LIN {X 0,Y 481.22,Z 200.296,A -85,B 0,C 180,E1 -6765.441,E2 -6765.441} C_VEL
LIN {X 0,Y 481.227,Z 196.018,A -85,B 0,C 180,E1 -6768.74,E2 -6768.74} C_VEL
LIN {X 0,Y 481.265,Z 192.611,A -85,B 0,C 180,E1 -6771.411,E2 -6771.411} C_VEL
LIN {X 0,Y 481.352,Z 189.237,A -85,B 0,C 180,E1 -6774.129,E2 -6774.129} C_VEL
LIN {X 0,Y 481.456,Z 185.54,A -85,B 0,C 180,E1 -6777.071,E2 -6777.071} C_VEL
LIN {X 0,Y 481.476,Z 183.514,A -85,B 0,C 180,E1 -6778.859,E2 -6778.859} C_VEL
LIN {X 0,Y 481.635,Z 183.493,A -85,B 0,C 180,E1 -6781.688,E2 -6781.688} C_VEL
LIN {X 0,Y 481.688,Z 183.482,A -85,B 0,C 180,E1 -6784.681,E2 -6784.681} C_VEL
LIN {X 0,Y 481.651,Z 183.487,A -85,B 0,C 180,E1 -6788.006,E2 -6788.006} C_VEL
LIN {X 0,Y 481.657,Z 183.49,A -85,B 0,C 180,E1 -6791.04,E2 -6791.04} C_VEL
LIN {X 0,Y 481.652,Z 183.484,A -85,B 0,C 180,E1 -6794.358,E2 -6794.358} C_VEL
LIN {X 0,Y 481.637,Z 183.492,A -85,B 0,C 180,E1 -6796.85,E2 -6796.85} C_VEL
LIN {X 0,Y 481.677,Z 183.481,A -85,B 0,C 180,E1 -6800.059,E2 -6800.059} C_VEL
LIN {X 0,Y 481.625,Z 183.488,A -85,B 0,C 180,E1 -6803.374,E2 -6803.374} C_VEL
LIN {X 0,Y 481.701,Z 183.482,A -85,B 0,C 180,E1 -6806.329,E2 -6806.329} C_VEL
LIN {X 0,Y 481.649,Z 183.484,A -85,B 0,C 180,E1 -6809.415,E2 -6809.415} C_VEL
LIN {X 0,Y 481.693,Z 183.485,A -85,B 0,C 180,E1 -6812.167,E2 -6812.167} C_VEL
LIN {X 0,Y 481.708,Z 183.474,A -85,B 0,C 180,E1 -6814.969,E2 -6814.969} C_VEL
LIN {X 0,Y 481.643,Z 183.49,A -85,B 0,C 180,E1 -6817.704,E2 -6817.704} C_VEL
LIN {X 0,Y 481.698,Z 183.479,A -85,B 0,C 180,E1 -6820.393,E2 -6820.393} C_VEL
LIN {X 0,Y 481.681,Z 183.482,A -85,B 0,C 180,E1 -6823.033,E2 -6823.033} C_VEL
LIN {X 0,Y 481.679,Z 183.484,A -85,B 0,C 180,E1 -6825.638,E2 -6825.638} C_VEL
LIN {X 0,Y 481.741,Z 183.473,A -85,B 0,C 180,E1 -6828.215,E2 -6828.215} C_VEL
LIN {X 0,Y 481.753,Z 183.476,A -85,B 0,C 180,E1 -6831.611,E2 -6831.611} C_VEL
LIN {X 0,Y 481.797,Z 183.464,A -85,B 0,C 180,E1 -6834.139,E2 -6834.139} C_VEL
LIN {X 0,Y 481.915,Z 183.454,A -85,B 0,C 180,E1 -6837.492,E2 -6837.492} C_VEL
LIN {X 0,Y 481.894,Z 183.456,A -85,B 0,C 180,E1 -6840.836,E2 -6840.836} C_VEL
LIN {X 0,Y 481.913,Z 183.455,A -85,B 0,C 180,E1 -6842.507,E2 -6842.507} C_VEL
LIN {X 0,Y 481.793,Z 183.466,A -85,B 0,C 180,E1 -6845.861,E2 -6845.861} C_VEL
LIN {X 0,Y 481.749,Z 183.478,A -85,B 0,C 180,E1 -6848.389,E2 -6848.389} C_VEL
LIN {X 0,Y 481.738,Z 183.475,A -85,B 0,C 180,E1 -6851.785,E2 -6851.785} C_VEL
LIN {X 0,Y 481.73,Z 183.475,A -85,B 0,C 180,E1 -6855.225,E2 -6855.225} C_VEL
LIN {X 0,Y 481.695,Z 183.481,A -85,B 0,C 180,E1 -6858.722,E2 -6858.722} C_VEL
LIN {X 0,Y 481.632,Z 183.489,A -85,B 0,C 180,E1 -6861.395,E2 -6861.395} C_VEL
LIN {X 0,Y 481.636,Z 183.493,A -85,B 0,C 180,E1 -6864.115,E2 -6864.115} C_VEL
LIN {X 0,Y 481.639,Z 183.489,A -85,B 0,C 180,E1 -6867.117,E2 -6867.117} C_VEL
LIN {X 0,Y 481.654,Z 183.491,A -85,B 0,C 180,E1 -6869.743,E2 -6869.743} C_VEL
LIN {X 0,Y 481.66,Z 183.484,A -85,B 0,C 180,E1 -6872.675,E2 -6872.675} C_VEL
LIN {X 0,Y 481.621,Z 183.493,A -85,B 0,C 180,E1 -6875.711,E2 -6875.711} C_VEL
LIN {X 0,Y 481.656,Z 183.491,A -85,B 0,C 180,E1 -6878.861,E2 -6878.861} C_VEL
LIN {X 0,Y 481.632,Z 183.489,A -85,B 0,C 180,E1 -6882.163,E2 -6882.163} C_VEL
LIN {X 0,Y 481.647,Z 183.488,A -85,B 0,C 180,E1 -6885.543,E2 -6885.543} C_VEL
LIN {X 0,Y 481.649,Z 183.492,A -85,B 0,C 180,E1 -6888.959,E2 -6888.959} C_VEL
LIN {X 0,Y 481.649,Z 183.49,A -85,B 0,C 180,E1 -6891.994,E2 -6891.994} C_VEL
LIN {X 0,Y 481.685,Z 183.481,A -85,B 0,C 180,E1 -6895.319,E2 -6895.319} C_VEL
LIN {X 0,Y 481.73,Z 183.66,A -85,B 0,C 180,E1 -6895.956,E2 -6895.956} C_VEL
LIN {X 0,Y 484.668,Z 196.394,A -85,B 0,C 180,E1 -6898.82,E2 -6898.82} C_VEL
LIN {X 0,Y 485.724,Z 201.979,A -85,B 0,C 180,E1 -6899.982,E2 -6899.982} C_VEL
LIN {X 0,Y 484.86,Z 216.213,A -85,B 0,C 180,E1 -6902.601,E2 -6902.601} C_VEL
LIN {X 0,Y 483.78,Z 235.626,A -85,B 0,C 180,E1 -6906,E2 -6906} C_VEL
LIN {X 0,Y 482.882,Z 255.103,A -85,B 0,C 180,E1 -6909.334,E2 -6909.334} C_VEL
LIN {X 0,Y 482.267,Z 271.753,A -85,B 0,C 180,E1 -6912.181,E2 -6912.181} C_VEL
LIN {X 0,Y 481.736,Z 289.457,A -85,B 0,C 180,E1 -6915.264,E2 -6915.264} C_VEL
LIN {X 0,Y 483.157,Z 305.726,A -85,B 0,C 180,E1 -6915.658,E2 -6915.658} C_VEL
LIN {X 0,Y 483.299,Z 312.328,A -85,B 0,C 180,E1 -6915.877,E2 -6915.877} C_VEL
LIN {X 0,Y 482.991,Z 325.423,A -85,B 0,C 180,E1 -6916.431,E2 -6916.431} C_VEL
LIN {X 0,Y 482.648,Z 336.61,A -85,B 0,C 180,E1 -6917.064,E2 -6917.064} C_VEL
LIN {X 0,Y 482.217,Z 348.057,A -85,B 0,C 180,E1 -6917.898,E2 -6917.898} C_VEL
LIN {X 0,Y 481.899,Z 358.618,A -85,B 0,C 180,E1 -6918.859,E2 -6918.859} C_VEL
LIN {X 0,Y 481.535,Z 368.02,A -85,B 0,C 180,E1 -6919.914,E2 -6919.914} C_VEL
LIN {X 0,Y 481.3,Z 377.093,A -85,B 0,C 180,E1 -6921.182,E2 -6921.182} C_VEL
LIN {X 0,Y 481.122,Z 384.382,A -85,B 0,C 180,E1 -6922.447,E2 -6922.447} C_VEL
LIN {X 0,Y 480.978,Z 390.38,A -85,B 0,C 180,E1 -6923.765,E2 -6923.765} C_VEL
LIN {X 0,Y 481.008,Z 394.686,A -85,B 0,C 180,E1 -6924.972,E2 -6924.972} C_VEL
LIN {X 0,Y 481.023,Z 397.058,A -85,B 0,C 180,E1 -6925.812,E2 -6925.812} C_VEL
LIN {X 0,Y 481.004,Z 398.985,A -85,B 0,C 180,E1 -6926.651,E2 -6926.651} C_VEL
LIN {X 0,Y 481.007,Z 400.451,A -85,B 0,C 180,E1 -6927.489,E2 -6927.489} C_VEL
LIN {X 0,Y 480.932,Z 402.075,A -85,B 0,C 180,E1 -6929.164,E2 -6929.164} C_VEL
LIN {X 0,Y 480.947,Z 402.282,A -85,B 0,C 180,E1 -6930.001,E2 -6930.001} C_VEL
LIN {X 0,Y 480.933,Z 402.03,A -85,B 0,C 180,E1 -6930.838,E2 -6930.838} C_VEL
LIN {X 0,Y 480.944,Z 401.367,A -85,B 0,C 180,E1 -6931.676,E2 -6931.676} C_VEL
LIN {X 0,Y 481.01,Z 400.303,A -85,B 0,C 180,E1 -6932.513,E2 -6932.513} C_VEL
LIN {X 0,Y 481.029,Z 398.792,A -85,B 0,C 180,E1 -6933.351,E2 -6933.351} C_VEL
LIN {X 0,Y 480.999,Z 395.665,A -85,B 0,C 180,E1 -6934.61,E2 -6934.61} C_VEL
LIN {X 0,Y 481.021,Z 391.432,A -85,B 0,C 180,E1 -6935.871,E2 -6935.871} C_VEL
LIN {X 0,Y 481.122,Z 384.92,A -85,B 0,C 180,E1 -6937.344,E2 -6937.344} C_VEL
LIN {X 0,Y 481.279,Z 377.82,A -85,B 0,C 180,E1 -6938.609,E2 -6938.609} C_VEL
LIN {X 0,Y 481.465,Z 368.907,A -85,B 0,C 180,E1 -6939.877,E2 -6939.877} C_VEL
LIN {X 0,Y 481.857,Z 358.791,A -85,B 0,C 180,E1 -6941.037,E2 -6941.037} C_VEL
LIN {X 0,Y 482.137,Z 347.375,A -85,B 0,C 180,E1 -6942.079,E2 -6942.079} C_VEL
LIN {X 0,Y 482.567,Z 335.494,A -85,B 0,C 180,E1 -6942.94,E2 -6942.94} C_VEL
LIN {X 0,Y 482.965,Z 323.218,A -85,B 0,C 180,E1 -6943.625,E2 -6943.625} C_VEL
LIN {X 0,Y 483.345,Z 309.934,A -85,B 0,C 180,E1 -6944.178,E2 -6944.178} C_VEL
LIN {X 0,Y 482.359,Z 295.934,A -85,B 0,C 180,E1 -6944.598,E2 -6944.598} C_VEL
LIN {X 0,Y 481.731,Z 289.296,A -85,B 0,C 180,E1 -6944.766,E2 -6944.766} C_VEL
LIN {X 0,Y 482.271,Z 270.473,A -85,B 0,C 180,E1 -6948.04,E2 -6948.04} C_VEL
LIN {X 0,Y 483.142,Z 250.047,A -85,B 0,C 180,E1 -6951.527,E2 -6951.527} C_VEL
LIN {X 0,Y 483.948,Z 231.674,A -85,B 0,C 180,E1 -6954.679,E2 -6954.679} C_VEL
LIN {X 0,Y 485.004,Z 213.512,A -85,B 0,C 180,E1 -6957.88,E2 -6957.88} C_VEL
LIN {X 0,Y 485.715,Z 201.921,A -85,B 0,C 180,E1 -6960.02,E2 -6960.02} C_VEL
LIN {X 0,Y 484.026,Z 193.683,A -85,B 0,C 180,E1 -6961.76,E2 -6961.76} C_VEL
LIN {X 0,Y 481.676,Z 183.492,A -85,B 0,C 180,E1 -6964.114,E2 -6964.114} C_VEL
LIN {X 0,Y 481.624,Z 183.496,A -85,B 0,C 180,E1 -6966.748,E2 -6966.748} C_VEL
LIN {X 0,Y 481.68,Z 183.486,A -85,B 0,C 180,E1 -6969.941,E2 -6969.941} C_VEL
LIN {X 0,Y 481.643,Z 183.49,A -85,B 0,C 180,E1 -6973.3,E2 -6973.3} C_VEL
LIN {X 0,Y 481.659,Z 183.491,A -85,B 0,C 180,E1 -6975.642,E2 -6975.642} C_VEL
LIN {X 0,Y 481.661,Z 183.491,A -85,B 0,C 180,E1 -6978.959,E2 -6978.959} C_VEL
LIN {X 0,Y 481.652,Z 183.49,A -85,B 0,C 180,E1 -6981.994,E2 -6981.994} C_VEL
LIN {X 0,Y 481.656,Z 183.504,A -85,B 0,C 180,E1 -6984.434,E2 -6984.434} C_VEL
LIN {X 0,Y 482.299,Z 187.95,A -85,B 0,C 180,E1 -6985.818,E2 -6985.818} C_VEL
LIN {X 0,Y 482.217,Z 196.061,A -85,B 0,C 180,E1 -6988.353,E2 -6988.353} C_VEL
LIN {X 0,Y 482.096,Z 206.422,A -85,B 0,C 180,E1 -6991.72,E2 -6991.72} C_VEL
LIN {X 0,Y 481.964,Z 215.165,A -85,B 0,C 180,E1 -6994.701,E2 -6994.701} C_VEL
LIN {X 0,Y 481.919,Z 222.689,A -85,B 0,C 180,E1 -6997.266,E2 -6997.266} C_VEL
LIN {X 0,Y 481.814,Z 231.6,A -85,B 0,C 180,E1 -7000.398,E2 -7000.398} C_VEL
LIN {X 0,Y 481.648,Z 241.418,A -85,B 0,C 180,E1 -7003.904,E2 -7003.904} C_VEL
LIN {X 0,Y 481.627,Z 244.929,A -85,B 0,C 180,E1 -7005.151,E2 -7005.151} C_VEL
LIN {X 0,Y 484.117,Z 257.015,A -85,B 0,C 180,E1 -7005.578,E2 -7005.578} C_VEL
LIN {X 0,Y 483.742,Z 270.706,A -85,B 0,C 180,E1 -7006.13,E2 -7006.13} C_VEL
LIN {X 0,Y 483.373,Z 283.042,A -85,B 0,C 180,E1 -7006.816,E2 -7006.816} C_VEL
LIN {X 0,Y 482.982,Z 295.454,A -85,B 0,C 180,E1 -7007.713,E2 -7007.713} C_VEL
LIN {X 0,Y 482.514,Z 305.818,A -85,B 0,C 180,E1 -7008.66,E2 -7008.66} C_VEL
LIN {X 0,Y 482.131,Z 315.197,A -85,B 0,C 180,E1 -7009.714,E2 -7009.714} C_VEL
LIN {X 0,Y 481.808,Z 322.924,A -85,B 0,C 180,E1 -7010.767,E2 -7010.767} C_VEL
LIN {X 0,Y 481.491,Z 330.49,A -85,B 0,C 180,E1 -7012.029,E2 -7012.029} C_VEL
LIN {X 0,Y 481.263,Z 337.504,A -85,B 0,C 180,E1 -7013.525,E2 -7013.525} C_VEL
LIN {X 0,Y 480.997,Z 342.655,A -85,B 0,C 180,E1 -7014.971,E2 -7014.971} C_VEL
LIN {X 0,Y 481.068,Z 344.937,A -85,B 0,C 180,E1 -7015.811,E2 -7015.811} C_VEL
LIN {X 0,Y 481.003,Z 346.806,A -85,B 0,C 180,E1 -7016.649,E2 -7016.649} C_VEL
LIN {X 0,Y 480.947,Z 348.246,A -85,B 0,C 180,E1 -7017.487,E2 -7017.487} C_VEL
LIN {X 0,Y 480.772,Z 349.845,A -85,B 0,C 180,E1 -7019.162,E2 -7019.162} C_VEL
LIN {X 0,Y 480.759,Z 350.06,A -85,B 0,C 180,E1 -7020,E2 -7020} C_VEL
LIN {X 0,Y 480.77,Z 349.843,A -85,B 0,C 180,E1 -7020.838,E2 -7020.838} C_VEL
LIN {X 0,Y 480.945,Z 348.202,A -85,B 0,C 180,E1 -7022.513,E2 -7022.513} C_VEL
LIN {X 0,Y 480.991,Z 346.783,A -85,B 0,C 180,E1 -7023.351,E2 -7023.351} C_VEL
LIN {X 0,Y 481.03,Z 343.822,A -85,B 0,C 180,E1 -7024.609,E2 -7024.609} C_VEL
LIN {X 0,Y 481.155,Z 339.808,A -85,B 0,C 180,E1 -7025.869,E2 -7025.869} C_VEL
LIN {X 0,Y 481.287,Z 334.625,A -85,B 0,C 180,E1 -7027.13,E2 -7027.13} C_VEL
LIN {X 0,Y 481.524,Z 328.112,A -85,B 0,C 180,E1 -7028.393,E2 -7028.393} C_VEL
LIN {X 0,Y 481.826,Z 320.026,A -85,B 0,C 180,E1 -7029.657,E2 -7029.657} C_VEL
LIN {X 0,Y 482.145,Z 311.758,A -85,B 0,C 180,E1 -7030.711,E2 -7030.711} C_VEL
LIN {X 0,Y 482.577,Z 301.598,A -85,B 0,C 180,E1 -7031.765,E2 -7031.765} C_VEL
LIN {X 0,Y 483.004,Z 290.302,A -85,B 0,C 180,E1 -7032.712,E2 -7032.712} C_VEL
LIN {X 0,Y 483.372,Z 279.109,A -85,B 0,C 180,E1 -7033.452,E2 -7033.452} C_VEL
LIN {X 0,Y 483.784,Z 266.716,A -85,B 0,C 180,E1 -7034.083,E2 -7034.083} C_VEL
LIN {X 0,Y 483.821,Z 255.619,A -85,B 0,C 180,E1 -7034.512,E2 -7034.512} C_VEL
LIN {X 0,Y 481.407,Z 243.352,A -85,B 0,C 180,E1 -7034.937,E2 -7034.937} C_VEL
LIN {X 0,Y 481.526,Z 235.352,A -85,B 0,C 180,E1 -7037.849,E2 -7037.849} C_VEL
LIN {X 0,Y 481.658,Z 226.855,A -85,B 0,C 180,E1 -7040.957,E2 -7040.957} C_VEL
LIN {X 0,Y 481.787,Z 219.5,A -85,B 0,C 180,E1 -7043.65,E2 -7043.65} C_VEL
LIN {X 0,Y 481.951,Z 210.681,A -85,B 0,C 180,E1 -7046.876,E2 -7046.876} C_VEL
LIN {X 0,Y 482.102,Z 202.963,A -85,B 0,C 180,E1 -7049.713,E2 -7049.713} C_VEL
LIN {X 0,Y 482.175,Z 195.007,A -85,B 0,C 180,E1 -7052.636,E2 -7052.636} C_VEL
LIN {X 0,Y 482.255,Z 187.65,A -85,B 0,C 180,E1 -7055.303,E2 -7055.303} C_VEL
LIN {X 0,Y 481.664,Z 183.489,A -85,B 0,C 180,E1 -7056.874,E2 -7056.874} C_VEL
LIN {X 0,Y 481.664,Z 183.487,A -85,B 0,C 180,E1 -7059.942,E2 -7059.942} C_VEL
LIN {X 0,Y 481.632,Z 183.491,A -85,B 0,C 180,E1 -7063.146,E2 -7063.146} C_VEL
LIN {X 0,Y 481.659,Z 183.487,A -85,B 0,C 180,E1 -7065.641,E2 -7065.641} C_VEL
LIN {X 0,Y 481.662,Z 183.49,A -85,B 0,C 180,E1 -7068.958,E2 -7068.958} C_VEL
LIN {X 0,Y 481.638,Z 183.492,A -85,B 0,C 180,E1 -7071.996,E2 -7071.996} C_VEL
LIN {X 0,Y 481.684,Z 183.488,A -85,B 0,C 180,E1 -7075.317,E2 -7075.317} C_VEL
LIN {X 0,Y 481.644,Z 183.49,A -85,B 0,C 180,E1 -7078.311,E2 -7078.311} C_VEL
LIN {X 0,Y 481.5,Z 183.509,A -85,B 0,C 180,E1 -7080.719,E2 -7080.719} C_VEL
LIN {X 0,Y 480.796,Z 183.851,A -85,B 0,C 180,E1 -7081.415,E2 -7081.415} C_VEL
LIN {X 0,Y 477.902,Z 185.342,A -85,B 0,C 180,E1 -7082.535,E2 -7082.535} C_VEL
LIN {X 0,Y 475.475,Z 186.77,A -85,B 0,C 180,E1 -7083.435,E2 -7083.435} C_VEL
LIN {X 0,Y 474.442,Z 187.776,A -85,B 0,C 180,E1 -7084.131,E2 -7084.131} C_VEL
LIN {X 0,Y 474.362,Z 188.066,A -85,B 0,C 180,E1 -7084.368,E2 -7084.368} C_VEL
LIN {X 0,Y 474.254,Z 191.754,A -85,B 0,C 180,E1 -7087.337,E2 -7087.337} C_VEL
LIN {X 0,Y 474.182,Z 195.164,A -85,B 0,C 180,E1 -7090.068,E2 -7090.068} C_VEL
LIN {X 0,Y 474.127,Z 198.642,A -85,B 0,C 180,E1 -7092.754,E2 -7092.754} C_VEL
LIN {X 0,Y 474.114,Z 202.159,A -85,B 0,C 180,E1 -7095.403,E2 -7095.403} C_VEL
LIN {X 0,Y 474.212,Z 205.883,A -85,B 0,C 180,E1 -7098.024,E2 -7098.024} C_VEL
LIN {X 0,Y 474.137,Z 209.896,A -85,B 0,C 180,E1 -7100.642,E2 -7100.642} C_VEL
LIN {X 0,Y 476.144,Z 219.9,A -85,B 0,C 180,E1 -7101.083,E2 -7101.083} C_VEL
LIN {X 0,Y 476.003,Z 228.87,A -85,B 0,C 180,E1 -7101.585,E2 -7101.585} C_VEL
LIN {X 0,Y 475.902,Z 236.501,A -85,B 0,C 180,E1 -7102.162,E2 -7102.162} C_VEL
LIN {X 0,Y 475.649,Z 242.928,A -85,B 0,C 180,E1 -7102.784,E2 -7102.784} C_VEL
LIN {X 0,Y 475.534,Z 249.697,A -85,B 0,C 180,E1 -7103.635,E2 -7103.635} C_VEL
LIN {X 0,Y 475.19,Z 255.993,A -85,B 0,C 180,E1 -7104.695,E2 -7104.695} C_VEL
LIN {X 0,Y 475.005,Z 260.57,A -85,B 0,C 180,E1 -7105.756,E2 -7105.756} C_VEL
LIN {X 0,Y 474.731,Z 264.378,A -85,B 0,C 180,E1 -7107.029,E2 -7107.029} C_VEL
LIN {X 0,Y 474.572,Z 266.665,A -85,B 0,C 180,E1 -7108.302,E2 -7108.302} C_VEL
LIN {X 0,Y 474.49,Z 267.471,A -85,B 0,C 180,E1 -7109.15,E2 -7109.15} C_VEL
LIN {X 0,Y 474.459,Z 267.751,A -85,B 0,C 180,E1 -7109.999,E2 -7109.999} C_VEL
LIN {X 0,Y 474.482,Z 267.526,A -85,B 0,C 180,E1 -7110.848,E2 -7110.848} C_VEL
LIN {X 0,Y 474.521,Z 266.784,A -85,B 0,C 180,E1 -7111.696,E2 -7111.696} C_VEL
LIN {X 0,Y 474.576,Z 265.484,A -85,B 0,C 180,E1 -7112.545,E2 -7112.545} C_VEL
LIN {X 0,Y 474.921,Z 262.316,A -85,B 0,C 180,E1 -7113.817,E2 -7113.817} C_VEL
LIN {X 0,Y 475.055,Z 257.48,A -85,B 0,C 180,E1 -7115.091,E2 -7115.091} C_VEL
LIN {X 0,Y 475.298,Z 253.005,A -85,B 0,C 180,E1 -7115.94,E2 -7115.94} C_VEL
LIN {X 0,Y 475.509,Z 247.232,A -85,B 0,C 180,E1 -7116.789,E2 -7116.789} C_VEL
LIN {X 0,Y 475.751,Z 240.766,A -85,B 0,C 180,E1 -7117.532,E2 -7117.532} C_VEL
LIN {X 0,Y 475.976,Z 232.3,A -85,B 0,C 180,E1 -7118.275,E2 -7118.275} C_VEL
LIN {X 0,Y 476.099,Z 222.919,A -85,B 0,C 180,E1 -7118.862,E2 -7118.862} C_VEL
LIN {X 0,Y 475.943,Z 218.408,A -85,B 0,C 180,E1 -7119.079,E2 -7119.079} C_VEL
LIN {X 0,Y 474.141,Z 209.92,A -85,B 0,C 180,E1 -7119.436,E2 -7119.436} C_VEL
LIN {X 0,Y 474.206,Z 205.991,A -85,B 0,C 180,E1 -7121.996,E2 -7121.996} C_VEL
LIN {X 0,Y 474.157,Z 201.011,A -85,B 0,C 180,E1 -7125.541,E2 -7125.541} C_VEL
LIN {X 0,Y 474.177,Z 196.488,A -85,B 0,C 180,E1 -7129.029,E2 -7129.029} C_VEL
LIN {X 0,Y 474.23,Z 193.027,A -85,B 0,C 180,E1 -7131.745,E2 -7131.745} C_VEL
LIN {X 0,Y 474.31,Z 189.602,A -85,B 0,C 180,E1 -7134.511,E2 -7134.511} C_VEL
LIN {X 0,Y 474.404,Z 186.065,A -85,B 0,C 180,E1 -7137.337,E2 -7137.337} C_VEL
LIN {X 0,Y 474.398,Z 184.851,A -85,B 0,C 180,E1 -7138.297,E2 -7138.297} C_VEL
LIN {X 0,Y 474.453,Z 184.389,A -85,B 0,C 180,E1 -7139.262,E2 -7139.262} C_VEL
LIN {X 0,Y 474.631,Z 184.362,A -85,B 0,C 180,E1 -7142.211,E2 -7142.211} C_VEL
LIN {X 0,Y 474.624,Z 184.366,A -85,B 0,C 180,E1 -7145.273,E2 -7145.273} C_VEL
LIN {X 0,Y 474.607,Z 184.363,A -85,B 0,C 180,E1 -7148.456,E2 -7148.456} C_VEL
LIN {X 0,Y 474.626,Z 184.365,A -85,B 0,C 180,E1 -7150.959,E2 -7150.959} C_VEL
LIN {X 0,Y 474.608,Z 184.361,A -85,B 0,C 180,E1 -7154.103,E2 -7154.103} C_VEL
LIN {X 0,Y 474.608,Z 184.369,A -85,B 0,C 180,E1 -7157.065,E2 -7157.065} C_VEL
LIN {X 0,Y 474.654,Z 184.359,A -85,B 0,C 180,E1 -7160.455,E2 -7160.455} C_VEL
LIN {X 0,Y 474.586,Z 184.364,A -85,B 0,C 180,E1 -7163.676,E2 -7163.676} C_VEL
LIN {X 0,Y 474.634,Z 184.363,A -85,B 0,C 180,E1 -7166.779,E2 -7166.779} C_VEL
LIN {X 0,Y 474.605,Z 184.363,A -85,B 0,C 180,E1 -7169.77,E2 -7169.77} C_VEL
LIN {X 0,Y 474.705,Z 184.352,A -85,B 0,C 180,E1 -7172.68,E2 -7172.68} C_VEL
LIN {X 0,Y 474.649,Z 184.354,A -85,B 0,C 180,E1 -7175.506,E2 -7175.506} C_VEL
LIN {X 0,Y 474.66,Z 184.354,A -85,B 0,C 180,E1 -7179.185,E2 -7179.185} C_VEL
LIN {X 0,Y 474.646,Z 184.364,A -85,B 0,C 180,E1 -7181.884,E2 -7181.884} C_VEL
LIN {X 0,Y 474.689,Z 184.347,A -85,B 0,C 180,E1 -7184.544,E2 -7184.544} C_VEL
LIN {X 0,Y 474.694,Z 184.352,A -85,B 0,C 180,E1 -7188.037,E2 -7188.037} C_VEL
LIN {X 0,Y 474.718,Z 184.354,A -85,B 0,C 180,E1 -7191.486,E2 -7191.486} C_VEL
LIN {X 0,Y 474.759,Z 184.341,A -85,B 0,C 180,E1 -7194.052,E2 -7194.052} C_VEL
LIN {X 0,Y 474.881,Z 184.331,A -85,B 0,C 180,E1 -7197.455,E2 -7197.455} C_VEL
LIN {X 0,Y 474.845,Z 184.333,A -85,B 0,C 180,E1 -7200.848,E2 -7200.848} C_VEL
LIN {X 0,Y 474.879,Z 184.332,A -85,B 0,C 180,E1 -7202.545,E2 -7202.545} C_VEL
LIN {X 0,Y 474.756,Z 184.342,A -85,B 0,C 180,E1 -7205.948,E2 -7205.948} C_VEL
LIN {X 0,Y 474.714,Z 184.353,A -85,B 0,C 180,E1 -7208.514,E2 -7208.514} C_VEL
LIN {X 0,Y 474.692,Z 184.354,A -85,B 0,C 180,E1 -7211.963,E2 -7211.963} C_VEL
LIN {X 0,Y 474.687,Z 184.353,A -85,B 0,C 180,E1 -7215.456,E2 -7215.456} C_VEL
LIN {X 0,Y 474.649,Z 184.358,A -85,B 0,C 180,E1 -7219.011,E2 -7219.011} C_VEL
LIN {X 0,Y 474.575,Z 184.372,A -85,B 0,C 180,E1 -7221.73,E2 -7221.73} C_VEL
LIN {X 0,Y 474.614,Z 184.364,A -85,B 0,C 180,E1 -7224.495,E2 -7224.495} C_VEL
LIN {X 0,Y 474.586,Z 184.369,A -85,B 0,C 180,E1 -7227.327,E2 -7227.327} C_VEL
LIN {X 0,Y 474.585,Z 184.367,A -85,B 0,C 180,E1 -7230.232,E2 -7230.232} C_VEL
LIN {X 0,Y 474.615,Z 184.366,A -85,B 0,C 180,E1 -7233.222,E2 -7233.222} C_VEL
LIN {X 0,Y 474.573,Z 184.368,A -85,B 0,C 180,E1 -7236.325,E2 -7236.325} C_VEL
LIN {X 0,Y 474.612,Z 184.362,A -85,B 0,C 180,E1 -7239.549,E2 -7239.549} C_VEL
LIN {X 0,Y 474.593,Z 184.373,A -85,B 0,C 180,E1 -7242.937,E2 -7242.937} C_VEL
LIN {X 0,Y 474.599,Z 184.365,A -85,B 0,C 180,E1 -7245.896,E2 -7245.896} C_VEL
LIN {X 0,Y 474.621,Z 184.368,A -85,B 0,C 180,E1 -7249.042,E2 -7249.042} C_VEL
LIN {X 0,Y 474.604,Z 184.366,A -85,B 0,C 180,E1 -7251.705,E2 -7251.705} C_VEL
LIN {X 0,Y 474.645,Z 184.357,A -85,B 0,C 180,E1 -7255.247,E2 -7255.247} C_VEL
LIN {X 0,Y 474.669,Z 184.503,A -85,B 0,C 180,E1 -7255.571,E2 -7255.571} C_VEL
LIN {X 0,Y 477.689,Z 197.53,A -85,B 0,C 180,E1 -7258.575,E2 -7258.575} C_VEL
LIN {X 0,Y 478.857,Z 204.207,A -85,B 0,C 180,E1 -7259.988,E2 -7259.988} C_VEL
LIN {X 0,Y 477.797,Z 219.719,A -85,B 0,C 180,E1 -7262.873,E2 -7262.873} C_VEL
LIN {X 0,Y 476.721,Z 238.948,A -85,B 0,C 180,E1 -7266.295,E2 -7266.295} C_VEL
LIN {X 0,Y 475.81,Z 257.117,A -85,B 0,C 180,E1 -7269.465,E2 -7269.465} C_VEL
LIN {X 0,Y 475.202,Z 272.337,A -85,B 0,C 180,E1 -7272.13,E2 -7272.13} C_VEL
LIN {X 0,Y 474.677,Z 288.639,A -85,B 0,C 180,E1 -7275.039,E2 -7275.039} C_VEL
LIN {X 0,Y 476.113,Z 305.083,A -85,B 0,C 180,E1 -7275.441,E2 -7275.441} C_VEL
LIN {X 0,Y 476.421,Z 310.244,A -85,B 0,C 180,E1 -7275.614,E2 -7275.614} C_VEL
LIN {X 0,Y 476.11,Z 322.658,A -85,B 0,C 180,E1 -7276.122,E2 -7276.122} C_VEL
LIN {X 0,Y 475.695,Z 334.327,A -85,B 0,C 180,E1 -7276.763,E2 -7276.763} C_VEL
LIN {X 0,Y 475.279,Z 345.747,A -85,B 0,C 180,E1 -7277.568,E2 -7277.568} C_VEL
LIN {X 0,Y 474.903,Z 357.049,A -85,B 0,C 180,E1 -7278.585,E2 -7278.585} C_VEL
LIN {X 0,Y 474.507,Z 367.551,A -85,B 0,C 180,E1 -7279.763,E2 -7279.763} C_VEL
LIN {X 0,Y 474.238,Z 376.641,A -85,B 0,C 180,E1 -7281.049,E2 -7281.049} C_VEL
LIN {X 0,Y 474.047,Z 383.947,A -85,B 0,C 180,E1 -7282.333,E2 -7282.333} C_VEL
LIN {X 0,Y 473.88,Z 390.444,A -85,B 0,C 180,E1 -7283.797,E2 -7283.797} C_VEL
LIN {X 0,Y 473.935,Z 394.285,A -85,B 0,C 180,E1 -7284.897,E2 -7284.897} C_VEL
LIN {X 0,Y 473.919,Z 396.66,A -85,B 0,C 180,E1 -7285.749,E2 -7285.749} C_VEL
LIN {X 0,Y 473.929,Z 398.592,A -85,B 0,C 180,E1 -7286.601,E2 -7286.601} C_VEL
LIN {X 0,Y 473.913,Z 400.064,A -85,B 0,C 180,E1 -7287.451,E2 -7287.451} C_VEL
LIN {X 0,Y 473.864,Z 401.078,A -85,B 0,C 180,E1 -7288.301,E2 -7288.301} C_VEL
LIN {X 0,Y 473.85,Z 401.69,A -85,B 0,C 180,E1 -7289.151,E2 -7289.151} C_VEL
LIN {X 0,Y 473.862,Z 401.897,A -85,B 0,C 180,E1 -7290.001,E2 -7290.001} C_VEL
LIN {X 0,Y 473.851,Z 401.643,A -85,B 0,C 180,E1 -7290.851,E2 -7290.851} C_VEL
LIN {X 0,Y 473.871,Z 400.976,A -85,B 0,C 180,E1 -7291.701,E2 -7291.701} C_VEL
LIN {X 0,Y 473.917,Z 399.906,A -85,B 0,C 180,E1 -7292.551,E2 -7292.551} C_VEL
LIN {X 0,Y 473.951,Z 398.389,A -85,B 0,C 180,E1 -7293.402,E2 -7293.402} C_VEL
LIN {X 0,Y 473.909,Z 395.248,A -85,B 0,C 180,E1 -7294.68,E2 -7294.68} C_VEL
LIN {X 0,Y 473.926,Z 391.004,A -85,B 0,C 180,E1 -7295.959,E2 -7295.959} C_VEL
LIN {X 0,Y 474.032,Z 384.484,A -85,B 0,C 180,E1 -7297.455,E2 -7297.455} C_VEL
LIN {X 0,Y 474.187,Z 377.374,A -85,B 0,C 180,E1 -7298.739,E2 -7298.739} C_VEL
LIN {X 0,Y 474.421,Z 368.448,A -85,B 0,C 180,E1 -7300.025,E2 -7300.025} C_VEL
LIN {X 0,Y 474.791,Z 358.34,A -85,B 0,C 180,E1 -7301.204,E2 -7301.204} C_VEL
LIN {X 0,Y 475.127,Z 347.527,A -85,B 0,C 180,E1 -7302.212,E2 -7302.212} C_VEL
LIN {X 0,Y 475.623,Z 335.135,A -85,B 0,C 180,E1 -7303.133,E2 -7303.133} C_VEL
LIN {X 0,Y 476.03,Z 322.94,A -85,B 0,C 180,E1 -7303.828,E2 -7303.828} C_VEL
LIN {X 0,Y 476.477,Z 309.85,A -85,B 0,C 180,E1 -7304.386,E2 -7304.386} C_VEL
LIN {X 0,Y 475.557,Z 297.058,A -85,B 0,C 180,E1 -7304.798,E2 -7304.798} C_VEL
LIN {X 0,Y 474.638,Z 288.331,A -85,B 0,C 180,E1 -7305.019,E2 -7305.019} C_VEL
LIN {X 0,Y 475.215,Z 271.074,A -85,B 0,C 180,E1 -7308.095,E2 -7308.095} C_VEL
LIN {X 0,Y 476.141,Z 251.09,A -85,B 0,C 180,E1 -7311.58,E2 -7311.58} C_VEL
LIN {X 0,Y 477.029,Z 232.531,A -85,B 0,C 180,E1 -7314.828,E2 -7314.828} C_VEL
LIN {X 0,Y 478.135,Z 214.582,A -85,B 0,C 180,E1 -7318.059,E2 -7318.059} C_VEL
LIN {X 0,Y 478.866,Z 204.169,A -85,B 0,C 180,E1 -7320.014,E2 -7320.014} C_VEL
LIN {X 0,Y 477.656,Z 197.516,A -85,B 0,C 180,E1 -7321.418,E2 -7321.418} C_VEL
LIN {X 0,Y 474.657,Z 184.366,A -85,B 0,C 180,E1 -7324.465,E2 -7324.465} C_VEL
LIN {X 0,Y 474.589,Z 184.37,A -85,B 0,C 180,E1 -7327.385,E2 -7327.385} C_VEL
LIN {X 0,Y 474.622,Z 184.365,A -85,B 0,C 180,E1 -7330.658,E2 -7330.658} C_VEL
LIN {X 0,Y 474.605,Z 184.368,A -85,B 0,C 180,E1 -7333.481,E2 -7333.481} C_VEL
LIN {X 0,Y 474.605,Z 184.366,A -85,B 0,C 180,E1 -7336.52,E2 -7336.52} C_VEL
LIN {X 0,Y 474.622,Z 184.367,A -85,B 0,C 180,E1 -7339.343,E2 -7339.343} C_VEL
LIN {X 0,Y 474.586,Z 184.372,A -85,B 0,C 180,E1 -7342.616,E2 -7342.616} C_VEL
LIN {X 0,Y 474.592,Z 184.487,A -85,B 0,C 180,E1 -7344.134,E2 -7344.134} C_VEL
LIN {X 0,Y 475.412,Z 189.891,A -85,B 0,C 180,E1 -7345.879,E2 -7345.879} C_VEL
LIN {X 0,Y 475.288,Z 197.637,A -85,B 0,C 180,E1 -7348.336,E2 -7348.336} C_VEL
LIN {X 0,Y 475.161,Z 208.018,A -85,B 0,C 180,E1 -7351.751,E2 -7351.751} C_VEL
LIN {X 0,Y 475.018,Z 217.708,A -85,B 0,C 180,E1 -7355.06,E2 -7355.06} C_VEL
LIN {X 0,Y 474.906,Z 225.621,A -85,B 0,C 180,E1 -7357.829,E2 -7357.829} C_VEL
LIN {X 0,Y 474.787,Z 234.518,A -85,B 0,C 180,E1 -7360.995,E2 -7360.995} C_VEL
LIN {X 0,Y 474.613,Z 243.581,A -85,B 0,C 180,E1 -7364.264,E2 -7364.264} C_VEL
LIN {X 0,Y 474.637,Z 245.305,A -85,B 0,C 180,E1 -7364.889,E2 -7364.889} C_VEL
LIN {X 0,Y 477.271,Z 257.931,A -85,B 0,C 180,E1 -7365.367,E2 -7365.367} C_VEL
LIN {X 0,Y 476.889,Z 271.415,A -85,B 0,C 180,E1 -7365.927,E2 -7365.927} C_VEL
LIN {X 0,Y 476.504,Z 283.815,A -85,B 0,C 180,E1 -7366.636,E2 -7366.636} C_VEL
LIN {X 0,Y 476.065,Z 295.96,A -85,B 0,C 180,E1 -7367.531,E2 -7367.531} C_VEL
LIN {X 0,Y 475.575,Z 306.282,A -85,B 0,C 180,E1 -7368.492,E2 -7368.492} C_VEL
LIN {X 0,Y 475.165,Z 315.653,A -85,B 0,C 180,E1 -7369.561,E2 -7369.561} C_VEL
LIN {X 0,Y 474.813,Z 323.363,A -85,B 0,C 180,E1 -7370.63,E2 -7370.63} C_VEL
LIN {X 0,Y 474.469,Z 330.917,A -85,B 0,C 180,E1 -7371.911,E2 -7371.911} C_VEL
LIN {X 0,Y 474.225,Z 336.945,A -85,B 0,C 180,E1 -7373.191,E2 -7373.191} C_VEL
LIN {X 0,Y 473.99,Z 341.718,A -85,B 0,C 180,E1 -7374.469,E2 -7374.469} C_VEL
LIN {X 0,Y 474.012,Z 345.353,A -85,B 0,C 180,E1 -7375.749,E2 -7375.749} C_VEL
LIN {X 0,Y 473.931,Z 347.218,A -85,B 0,C 180,E1 -7376.599,E2 -7376.599} C_VEL
LIN {X 0,Y 473.888,Z 348.652,A -85,B 0,C 180,E1 -7377.45,E2 -7377.45} C_VEL
LIN {X 0,Y 473.7,Z 350.241,A -85,B 0,C 180,E1 -7379.15,E2 -7379.15} C_VEL
LIN {X 0,Y 473.685,Z 350.45,A -85,B 0,C 180,E1 -7380,E2 -7380} C_VEL
LIN {X 0,Y 473.698,Z 350.223,A -85,B 0,C 180,E1 -7380.85,E2 -7380.85} C_VEL
LIN {X 0,Y 473.886,Z 348.565,A -85,B 0,C 180,E1 -7382.55,E2 -7382.55} C_VEL
LIN {X 0,Y 473.919,Z 347.133,A -85,B 0,C 180,E1 -7383.401,E2 -7383.401} C_VEL
LIN {X 0,Y 473.947,Z 344.153,A -85,B 0,C 180,E1 -7384.678,E2 -7384.678} C_VEL
LIN {X 0,Y 474.114,Z 340.113,A -85,B 0,C 180,E1 -7385.956,E2 -7385.956} C_VEL
LIN {X 0,Y 474.261,Z 333.904,A -85,B 0,C 180,E1 -7387.45,E2 -7387.45} C_VEL
LIN {X 0,Y 474.548,Z 327.141,A -85,B 0,C 180,E1 -7388.731,E2 -7388.731} C_VEL
LIN {X 0,Y 474.892,Z 318.682,A -85,B 0,C 180,E1 -7390.014,E2 -7390.014} C_VEL
LIN {X 0,Y 475.237,Z 310.023,A -85,B 0,C 180,E1 -7391.084,E2 -7391.084} C_VEL
LIN {X 0,Y 475.76,Z 299.436,A -85,B 0,C 180,E1 -7392.152,E2 -7392.152} C_VEL
LIN {X 0,Y 476.087,Z 288.756,A -85,B 0,C 180,E1 -7393.017,E2 -7393.017} C_VEL
LIN {X 0,Y 476.522,Z 277.238,A -85,B 0,C 180,E1 -7393.758,E2 -7393.758} C_VEL
LIN {X 0,Y 476.942,Z 265.458,A -85,B 0,C 180,E1 -7394.344,E2 -7394.344} C_VEL
LIN {X 0,Y 476.872,Z 256.215,A -85,B 0,C 180,E1 -7394.701,E2 -7394.701} C_VEL
LIN {X 0,Y 474.375,Z 243.679,A -85,B 0,C 180,E1 -7395.137,E2 -7395.137} C_VEL
LIN {X 0,Y 474.502,Z 235.523,A -85,B 0,C 180,E1 -7398.122,E2 -7398.122} C_VEL
LIN {X 0,Y 474.63,Z 227.379,A -85,B 0,C 180,E1 -7401.113,E2 -7401.113} C_VEL
LIN {X 0,Y 474.769,Z 219.481,A -85,B 0,C 180,E1 -7404.022,E2 -7404.022} C_VEL
LIN {X 0,Y 474.96,Z 210.33,A -85,B 0,C 180,E1 -7407.398,E2 -7407.398} C_VEL
LIN {X 0,Y 475.129,Z 202.732,A -85,B 0,C 180,E1 -7410.194,E2 -7410.194} C_VEL
LIN {X 0,Y 475.221,Z 194.633,A -85,B 0,C 180,E1 -7413.175,E2 -7413.175} C_VEL
LIN {X 0,Y 475.205,Z 188.137,A -85,B 0,C 180,E1 -7415.568,E2 -7415.568} C_VEL
LIN {X 0,Y 474.632,Z 184.365,A -85,B 0,C 180,E1 -7417.004,E2 -7417.004} C_VEL
LIN {X 0,Y 474.613,Z 184.368,A -85,B 0,C 180,E1 -7419.644,E2 -7419.644} C_VEL
LIN {X 0,Y 474.605,Z 184.367,A -85,B 0,C 180,E1 -7422.233,E2 -7422.233} C_VEL
LIN {X 0,Y 474.622,Z 184.362,A -85,B 0,C 180,E1 -7425.297,E2 -7425.297} C_VEL
LIN {X 0,Y 474.626,Z 184.363,A -85,B 0,C 180,E1 -7428.214,E2 -7428.214} C_VEL
LIN {X 0,Y 474.635,Z 184.365,A -85,B 0,C 180,E1 -7430.452,E2 -7430.452} C_VEL
LIN {X 0,Y 474.577,Z 184.373,A -85,B 0,C 180,E1 -7433.674,E2 -7433.674} C_VEL
LIN {X 0,Y 474.627,Z 184.365,A -85,B 0,C 180,E1 -7436.778,E2 -7436.778} C_VEL
LIN {X 0,Y 474.532,Z 184.376,A -85,B 0,C 180,E1 -7439.764,E2 -7439.764} C_VEL
LIN {X 0,Y 474.452,Z 184.389,A -85,B 0,C 180,E1 -7440.923,E2 -7440.923} C_VEL
LIN {X 0,Y 474.399,Z 184.736,A -85,B 0,C 180,E1 -7441.701,E2 -7441.701} C_VEL
LIN {X 0,Y 474.362,Z 188.066,A -85,B 0,C 180,E1 -7444.368,E2 -7444.368} C_VEL
LIN {X 0,Y 473.699,Z 189.02,A -85,B 0,C 180,E1 -7445.067,E2 -7445.067} C_VEL
LIN {X 0,Y 470.808,Z 190.769,A -85,B 0,C 180,E1 -7446.199,E2 -7446.199} C_VEL
LIN {X 0,Y 468.345,Z 192.185,A -85,B 0,C 180,E1 -7447.11,E2 -7447.11} C_VEL
LIN {X 0,Y 467.272,Z 193.186,A -85,B 0,C 180,E1 -7447.817,E2 -7447.817} C_VEL
LIN {X 0,Y 467.177,Z 193.497,A -85,B 0,C 180,E1 -7448.057,E2 -7448.057} C_VEL
LIN {X 0,Y 467.149,Z 197.947,A -85,B 0,C 180,E1 -7451.582,E2 -7451.582} C_VEL
LIN {X 0,Y 467.099,Z 202.711,A -85,B 0,C 180,E1 -7455.179,E2 -7455.179} C_VEL
LIN {X 0,Y 467.126,Z 207.793,A -85,B 0,C 180,E1 -7458.72,E2 -7458.72} C_VEL
LIN {X 0,Y 467.061,Z 210.524,A -85,B 0,C 180,E1 -7460.472,E2 -7460.472} C_VEL
LIN {X 0,Y 469.176,Z 220.362,A -85,B 0,C 180,E1 -7460.895,E2 -7460.895} C_VEL
LIN {X 0,Y 469.089,Z 229.788,A -85,B 0,C 180,E1 -7461.429,E2 -7461.429} C_VEL
LIN {X 0,Y 469.008,Z 236.409,A -85,B 0,C 180,E1 -7461.93,E2 -7461.93} C_VEL
LIN {X 0,Y 468.739,Z 243.096,A -85,B 0,C 180,E1 -7462.569,E2 -7462.569} C_VEL
LIN {X 0,Y 468.627,Z 249.271,A -85,B 0,C 180,E1 -7463.325,E2 -7463.325} C_VEL
LIN {X 0,Y 468.387,Z 254.782,A -85,B 0,C 180,E1 -7464.186,E2 -7464.186} C_VEL
LIN {X 0,Y 468.025,Z 259.956,A -85,B 0,C 180,E1 -7465.262,E2 -7465.262} C_VEL
LIN {X 0,Y 467.82,Z 264.297,A -85,B 0,C 180,E1 -7466.554,E2 -7466.554} C_VEL
LIN {X 0,Y 467.569,Z 266.299,A -85,B 0,C 180,E1 -7467.414,E2 -7467.414} C_VEL
LIN {X 0,Y 467.558,Z 267.647,A -85,B 0,C 180,E1 -7468.276,E2 -7468.276} C_VEL
LIN {X 0,Y 467.471,Z 268.447,A -85,B 0,C 180,E1 -7469.137,E2 -7469.137} C_VEL
LIN {X 0,Y 467.438,Z 268.724,A -85,B 0,C 180,E1 -7469.999,E2 -7469.999} C_VEL
LIN {X 0,Y 467.463,Z 268.5,A -85,B 0,C 180,E1 -7470.86,E2 -7470.86} C_VEL
LIN {X 0,Y 467.511,Z 267.762,A -85,B 0,C 180,E1 -7471.722,E2 -7471.722} C_VEL
LIN {X 0,Y 467.563,Z 266.471,A -85,B 0,C 180,E1 -7472.583,E2 -7472.583} C_VEL
LIN {X 0,Y 467.935,Z 263.321,A -85,B 0,C 180,E1 -7473.874,E2 -7473.874} C_VEL
LIN {X 0,Y 468.062,Z 258.525,A -85,B 0,C 180,E1 -7475.168,E2 -7475.168} C_VEL
LIN {X 0,Y 468.321,Z 254.091,A -85,B 0,C 180,E1 -7476.029,E2 -7476.029} C_VEL
LIN {X 0,Y 468.55,Z 248.358,A -85,B 0,C 180,E1 -7476.891,E2 -7476.891} C_VEL
LIN {X 0,Y 468.815,Z 241.943,A -85,B 0,C 180,E1 -7477.644,E2 -7477.644} C_VEL
LIN {X 0,Y 469.045,Z 233.705,A -85,B 0,C 180,E1 -7478.39,E2 -7478.39} C_VEL
LIN {X 0,Y 469.175,Z 225.36,A -85,B 0,C 180,E1 -7478.939,E2 -7478.939} C_VEL
LIN {X 0,Y 469.118,Z 220.055,A -85,B 0,C 180,E1 -7479.212,E2 -7479.212} C_VEL
LIN {X 0,Y 467.095,Z 210.502,A -85,B 0,C 180,E1 -7479.635,E2 -7479.635} C_VEL
LIN {X 0,Y 467.133,Z 206.632,A -85,B 0,C 180,E1 -7482.158,E2 -7482.158} C_VEL
LIN {X 0,Y 467.111,Z 201.64,A -85,B 0,C 180,E1 -7485.712,E2 -7485.712} C_VEL
LIN {X 0,Y 467.135,Z 196.959,A -85,B 0,C 180,E1 -7489.327,E2 -7489.327} C_VEL
LIN {X 0,Y 467.18,Z 193.445,A -85,B 0,C 180,E1 -7492.09,E2 -7492.09} C_VEL
LIN {X 0,Y 467.268,Z 189.971,A -85,B 0,C 180,E1 -7494.905,E2 -7494.905} C_VEL
LIN {X 0,Y 467.357,Z 186.381,A -85,B 0,C 180,E1 -7497.784,E2 -7497.784} C_VEL
LIN {X 0,Y 467.349,Z 185.274,A -85,B 0,C 180,E1 -7498.763,E2 -7498.763} C_VEL
LIN {X 0,Y 467.573,Z 185.245,A -85,B 0,C 180,E1 -7501.739,E2 -7501.739} C_VEL
LIN {X 0,Y 467.563,Z 185.242,A -85,B 0,C 180,E1 -7504.831,E2 -7504.831} C_VEL
LIN {X 0,Y 467.56,Z 185.242,A -85,B 0,C 180,E1 -7508.043,E2 -7508.043} C_VEL
LIN {X 0,Y 467.576,Z 185.244,A -85,B 0,C 180,E1 -7511.276,E2 -7511.276} C_VEL
LIN {X 0,Y 467.56,Z 185.24,A -85,B 0,C 180,E1 -7513.821,E2 -7513.821} C_VEL
LIN {X 0,Y 467.549,Z 185.242,A -85,B 0,C 180,E1 -7516.255,E2 -7516.255} C_VEL
LIN {X 0,Y 467.571,Z 185.245,A -85,B 0,C 180,E1 -7518.722,E2 -7518.722} C_VEL
LIN {X 0,Y 467.559,Z 185.241,A -85,B 0,C 180,E1 -7521.955,E2 -7521.955} C_VEL
LIN {X 0,Y 467.56,Z 185.24,A -85,B 0,C 180,E1 -7525.167,E2 -7525.167} C_VEL
LIN {X 0,Y 467.577,Z 185.243,A -85,B 0,C 180,E1 -7528.259,E2 -7528.259} C_VEL
LIN {X 0,Y 467.574,Z 185.237,A -85,B 0,C 180,E1 -7531.25,E2 -7531.25} C_VEL
LIN {X 0,Y 467.602,Z 185.237,A -85,B 0,C 180,E1 -7534.159,E2 -7534.159} C_VEL
LIN {X 0,Y 467.567,Z 185.239,A -85,B 0,C 180,E1 -7536.995,E2 -7536.995} C_VEL
LIN {X 0,Y 467.613,Z 185.235,A -85,B 0,C 180,E1 -7539.777,E2 -7539.777} C_VEL
LIN {X 0,Y 467.599,Z 185.236,A -85,B 0,C 180,E1 -7542.506,E2 -7542.506} C_VEL
LIN {X 0,Y 467.595,Z 185.233,A -85,B 0,C 180,E1 -7545.196,E2 -7545.196} C_VEL
LIN {X 0,Y 467.645,Z 185.232,A -85,B 0,C 180,E1 -7547.854,E2 -7547.854} C_VEL
LIN {X 0,Y 467.671,Z 185.229,A -85,B 0,C 180,E1 -7551.357,E2 -7551.357} C_VEL
LIN {X 0,Y 467.724,Z 185.217,A -85,B 0,C 180,E1 -7553.962,E2 -7553.962} C_VEL
LIN {X 0,Y 467.847,Z 185.207,A -85,B 0,C 180,E1 -7557.417,E2 -7557.417} C_VEL
LIN {X 0,Y 467.868,Z 185.196,A -85,B 0,C 180,E1 -7560,E2 -7560} C_VEL
LIN {X 0,Y 467.845,Z 185.208,A -85,B 0,C 180,E1 -7562.583,E2 -7562.583} C_VEL
LIN {X 0,Y 467.721,Z 185.219,A -85,B 0,C 180,E1 -7566.038,E2 -7566.038} C_VEL
LIN {X 0,Y 467.667,Z 185.229,A -85,B 0,C 180,E1 -7568.643,E2 -7568.643} C_VEL
LIN {X 0,Y 467.641,Z 185.235,A -85,B 0,C 180,E1 -7572.358,E2 -7572.358} C_VEL
LIN {X 0,Y 467.637,Z 185.234,A -85,B 0,C 180,E1 -7575.885,E2 -7575.885} C_VEL
LIN {X 0,Y 467.609,Z 185.235,A -85,B 0,C 180,E1 -7579.308,E2 -7579.308} C_VEL
LIN {X 0,Y 467.518,Z 185.252,A -85,B 0,C 180,E1 -7582.075,E2 -7582.075} C_VEL
LIN {X 0,Y 467.547,Z 185.243,A -85,B 0,C 180,E1 -7584.891,E2 -7584.891} C_VEL
LIN {X 0,Y 467.532,Z 185.251,A -85,B 0,C 180,E1 -7587.775,E2 -7587.775} C_VEL
LIN {X 0,Y 467.554,Z 185.244,A -85,B 0,C 180,E1 -7591.045,E2 -7591.045} C_VEL
LIN {X 0,Y 467.567,Z 185.238,A -85,B 0,C 180,E1 -7594.241,E2 -7594.241} C_VEL
LIN {X 0,Y 467.532,Z 185.249,A -85,B 0,C 180,E1 -7597.186,E2 -7597.186} C_VEL
LIN {X 0,Y 467.55,Z 185.239,A -85,B 0,C 180,E1 -7600.268,E2 -7600.268} C_VEL
LIN {X 0,Y 467.552,Z 185.245,A -85,B 0,C 180,E1 -7602.564,E2 -7602.564} C_VEL
LIN {X 0,Y 467.558,Z 185.245,A -85,B 0,C 180,E1 -7605.054,E2 -7605.054} C_VEL
LIN {X 0,Y 467.582,Z 185.234,A -85,B 0,C 180,E1 -7607.441,E2 -7607.441} C_VEL
LIN {X 0,Y 467.576,Z 185.239,A -85,B 0,C 180,E1 -7610.857,E2 -7610.857} C_VEL
LIN {X 0,Y 467.554,Z 185.248,A -85,B 0,C 180,E1 -7614.262,E2 -7614.262} C_VEL
LIN {X 0,Y 467.624,Z 185.286,A -85,B 0,C 180,E1 -7615.174,E2 -7615.174} C_VEL
LIN {X 0,Y 470.713,Z 198.668,A -85,B 0,C 180,E1 -7618.325,E2 -7618.325} C_VEL
LIN {X 0,Y 471.996,Z 205.069,A -85,B 0,C 180,E1 -7619.726,E2 -7619.726} C_VEL
LIN {X 0,Y 471.172,Z 217.008,A -85,B 0,C 180,E1 -7622.005,E2 -7622.005} C_VEL
LIN {X 0,Y 470.052,Z 233.445,A -85,B 0,C 180,E1 -7625.016,E2 -7625.016} C_VEL
LIN {X 0,Y 469.262,Z 248.833,A -85,B 0,C 180,E1 -7627.782,E2 -7627.782} C_VEL
LIN {X 0,Y 468.424,Z 266.617,A -85,B 0,C 180,E1 -7630.948,E2 -7630.948} C_VEL
LIN {X 0,Y 467.683,Z 285.122,A -85,B 0,C 180,E1 -7634.308,E2 -7634.308} C_VEL
LIN {X 0,Y 467.602,Z 287.817,A -85,B 0,C 180,E1 -7634.808,E2 -7634.808} C_VEL
LIN {X 0,Y 468.906,Z 302.066,A -85,B 0,C 180,E1 -7635.156,E2 -7635.156} C_VEL
LIN {X 0,Y 469.461,Z 310.95,A -85,B 0,C 180,E1 -7635.451,E2 -7635.451} C_VEL
LIN {X 0,Y 469.117,Z 324.126,A -85,B 0,C 180,E1 -7636.022,E2 -7636.022} C_VEL
LIN {X 0,Y 468.689,Z 335.397,A -85,B 0,C 180,E1 -7636.672,E2 -7636.672} C_VEL
LIN {X 0,Y 468.255,Z 346.272,A -85,B 0,C 180,E1 -7637.473,E2 -7637.473} C_VEL
LIN {X 0,Y 467.846,Z 357.566,A -85,B 0,C 180,E1 -7638.52,E2 -7638.52} C_VEL
LIN {X 0,Y 467.482,Z 367.045,A -85,B 0,C 180,E1 -7639.608,E2 -7639.608} C_VEL
LIN {X 0,Y 467.192,Z 376.165,A -85,B 0,C 180,E1 -7640.913,E2 -7640.913} C_VEL
LIN {X 0,Y 466.967,Z 383.493,A -85,B 0,C 180,E1 -7642.216,E2 -7642.216} C_VEL
LIN {X 0,Y 466.848,Z 389.265,A -85,B 0,C 180,E1 -7643.503,E2 -7643.503} C_VEL
LIN {X 0,Y 466.861,Z 393.876,A -85,B 0,C 180,E1 -7644.819,E2 -7644.819} C_VEL
LIN {X 0,Y 466.818,Z 396.255,A -85,B 0,C 180,E1 -7645.684,E2 -7645.684} C_VEL
LIN {X 0,Y 466.855,Z 398.194,A -85,B 0,C 180,E1 -7646.549,E2 -7646.549} C_VEL
LIN {X 0,Y 466.823,Z 399.673,A -85,B 0,C 180,E1 -7647.413,E2 -7647.413} C_VEL
LIN {X 0,Y 466.794,Z 400.691,A -85,B 0,C 180,E1 -7648.276,E2 -7648.276} C_VEL
LIN {X 0,Y 466.771,Z 401.303,A -85,B 0,C 180,E1 -7649.138,E2 -7649.138} C_VEL
LIN {X 0,Y 466.78,Z 401.511,A -85,B 0,C 180,E1 -7650.001,E2 -7650.001} C_VEL
LIN {X 0,Y 466.773,Z 401.258,A -85,B 0,C 180,E1 -7650.864,E2 -7650.864} C_VEL
LIN {X 0,Y 466.801,Z 400.591,A -85,B 0,C 180,E1 -7651.727,E2 -7651.727} C_VEL
LIN {X 0,Y 466.828,Z 399.515,A -85,B 0,C 180,E1 -7652.59,E2 -7652.59} C_VEL
LIN {X 0,Y 466.841,Z 397.055,A -85,B 0,C 180,E1 -7653.886,E2 -7653.886} C_VEL
LIN {X 0,Y 466.866,Z 393.555,A -85,B 0,C 180,E1 -7655.183,E2 -7655.183} C_VEL
LIN {X 0,Y 466.873,Z 388.758,A -85,B 0,C 180,E1 -7656.524,E2 -7656.524} C_VEL
LIN {X 0,Y 467.012,Z 381.86,A -85,B 0,C 180,E1 -7658.003,E2 -7658.003} C_VEL
LIN {X 0,Y 467.235,Z 374.198,A -85,B 0,C 180,E1 -7659.307,E2 -7659.307} C_VEL
LIN {X 0,Y 467.448,Z 366.387,A -85,B 0,C 180,E1 -7660.395,E2 -7660.395} C_VEL
LIN {X 0,Y 467.877,Z 355.813,A -85,B 0,C 180,E1 -7661.591,E2 -7661.591} C_VEL
LIN {X 0,Y 468.213,Z 344.822,A -85,B 0,C 180,E1 -7662.597,E2 -7662.597} C_VEL
LIN {X 0,Y 468.76,Z 333.168,A -85,B 0,C 180,E1 -7663.439,E2 -7663.439} C_VEL
LIN {X 0,Y 469.245,Z 320.656,A -85,B 0,C 180,E1 -7664.142,E2 -7664.142} C_VEL
LIN {X 0,Y 469.444,Z 308.073,A -85,B 0,C 180,E1 -7664.676,E2 -7664.676} C_VEL
LIN {X 0,Y 468.377,Z 293.666,A -85,B 0,C 180,E1 -7665.128,E2 -7665.128} C_VEL
LIN {X 0,Y 467.615,Z 287.213,A -85,B 0,C 180,E1 -7665.306,E2 -7665.306} C_VEL
LIN {X 0,Y 468.242,Z 270.388,A -85,B 0,C 180,E1 -7668.374,E2 -7668.374} C_VEL
LIN {X 0,Y 469.146,Z 251.446,A -85,B 0,C 180,E1 -7671.753,E2 -7671.753} C_VEL
LIN {X 0,Y 470.094,Z 233.38,A -85,B 0,C 180,E1 -7674.984,E2 -7674.984} C_VEL
LIN {X 0,Y 471.179,Z 216.96,A -85,B 0,C 180,E1 -7677.997,E2 -7677.997} C_VEL
LIN {X 0,Y 471.977,Z 206.969,A -85,B 0,C 180,E1 -7679.896,E2 -7679.896} C_VEL
LIN {X 0,Y 471.658,Z 203.126,A -85,B 0,C 180,E1 -7680.688,E2 -7680.688} C_VEL
LIN {X 0,Y 469.043,Z 191.693,A -85,B 0,C 180,E1 -7683.273,E2 -7683.273} C_VEL
LIN {X 0,Y 467.616,Z 185.243,A -85,B 0,C 180,E1 -7684.895,E2 -7684.895} C_VEL
LIN {X 0,Y 467.562,Z 185.246,A -85,B 0,C 180,E1 -7688.591,E2 -7688.591} C_VEL
LIN {X 0,Y 467.582,Z 185.24,A -85,B 0,C 180,E1 -7691.403,E2 -7691.403} C_VEL
LIN {X 0,Y 467.557,Z 185.246,A -85,B 0,C 180,E1 -7693.821,E2 -7693.821} C_VEL
LIN {X 0,Y 467.559,Z 185.244,A -85,B 0,C 180,E1 -7696.256,E2 -7696.256} C_VEL
LIN {X 0,Y 467.583,Z 185.243,A -85,B 0,C 180,E1 -7698.724,E2 -7698.724} C_VEL
LIN {X 0,Y 467.565,Z 185.246,A -85,B 0,C 180,E1 -7701.955,E2 -7701.955} C_VEL
LIN {X 0,Y 467.589,Z 185.44,A -85,B 0,C 180,E1 -7703.78,E2 -7703.78} C_VEL
LIN {X 0,Y 468.506,Z 190.904,A -85,B 0,C 180,E1 -7705.594,E2 -7705.594} C_VEL
LIN {X 0,Y 468.409,Z 197.836,A -85,B 0,C 180,E1 -7707.816,E2 -7707.816} C_VEL
LIN {X 0,Y 468.195,Z 208.184,A -85,B 0,C 180,E1 -7711.292,E2 -7711.292} C_VEL
LIN {X 0,Y 468.064,Z 216.817,A -85,B 0,C 180,E1 -7714.278,E2 -7714.278} C_VEL
LIN {X 0,Y 467.995,Z 224.682,A -85,B 0,C 180,E1 -7717.018,E2 -7717.018} C_VEL
LIN {X 0,Y 467.819,Z 233.722,A -85,B 0,C 180,E1 -7720.244,E2 -7720.244} C_VEL
LIN {X 0,Y 467.669,Z 242.45,A -85,B 0,C 180,E1 -7723.41,E2 -7723.41} C_VEL
LIN {X 0,Y 467.644,Z 245.994,A -85,B 0,C 180,E1 -7724.64,E2 -7724.64} C_VEL
LIN {X 0,Y 470.385,Z 258.324,A -85,B 0,C 180,E1 -7725.12,E2 -7725.12} C_VEL
LIN {X 0,Y 470.108,Z 271.136,A -85,B 0,C 180,E1 -7725.664,E2 -7725.664} C_VEL
LIN {X 0,Y 469.687,Z 283.159,A -85,B 0,C 180,E1 -7726.347,E2 -7726.347} C_VEL
LIN {X 0,Y 469.226,Z 295.219,A -85,B 0,C 180,E1 -7727.237,E2 -7727.237} C_VEL
LIN {X 0,Y 468.69,Z 305.807,A -85,B 0,C 180,E1 -7728.211,E2 -7728.211} C_VEL
LIN {X 0,Y 468.269,Z 314.449,A -85,B 0,C 180,E1 -7729.187,E2 -7729.187} C_VEL
LIN {X 0,Y 467.828,Z 323.842,A -85,B 0,C 180,E1 -7730.488,E2 -7730.488} C_VEL
LIN {X 0,Y 467.446,Z 331.374,A -85,B 0,C 180,E1 -7731.788,E2 -7731.788} C_VEL
LIN {X 0,Y 467.185,Z 337.656,A -85,B 0,C 180,E1 -7733.152,E2 -7733.152} C_VEL
LIN {X 0,Y 466.945,Z 342.159,A -85,B 0,C 180,E1 -7734.386,E2 -7734.386} C_VEL
LIN {X 0,Y 466.958,Z 345.781,A -85,B 0,C 180,E1 -7735.684,E2 -7735.684} C_VEL
LIN {X 0,Y 466.862,Z 347.642,A -85,B 0,C 180,E1 -7736.548,E2 -7736.548} C_VEL
LIN {X 0,Y 466.831,Z 349.065,A -85,B 0,C 180,E1 -7737.411,E2 -7737.411} C_VEL
LIN {X 0,Y 466.63,Z 350.64,A -85,B 0,C 180,E1 -7739.137,E2 -7739.137} C_VEL
LIN {X 0,Y 466.613,Z 350.842,A -85,B 0,C 180,E1 -7740,E2 -7740} C_VEL
LIN {X 0,Y 466.629,Z 350.602,A -85,B 0,C 180,E1 -7740.863,E2 -7740.863} C_VEL
LIN {X 0,Y 466.799,Z 348.923,A -85,B 0,C 180,E1 -7742.589,E2 -7742.589} C_VEL
LIN {X 0,Y 466.849,Z 347.473,A -85,B 0,C 180,E1 -7743.452,E2 -7743.452} C_VEL
LIN {X 0,Y 466.871,Z 344.469,A -85,B 0,C 180,E1 -7744.749,E2 -7744.749} C_VEL
LIN {X 0,Y 467.068,Z 340.398,A -85,B 0,C 180,E1 -7746.046,E2 -7746.046} C_VEL
LIN {X 0,Y 467.217,Z 334.154,A -85,B 0,C 180,E1 -7747.563,E2 -7747.563} C_VEL
LIN {X 0,Y 467.535,Z 327.355,A -85,B 0,C 180,E1 -7748.863,E2 -7748.863} C_VEL
LIN {X 0,Y 467.882,Z 318.843,A -85,B 0,C 180,E1 -7750.166,E2 -7750.166} C_VEL
LIN {X 0,Y 468.281,Z 310.139,A -85,B 0,C 180,E1 -7751.251,E2 -7751.251} C_VEL
LIN {X 0,Y 468.808,Z 299.489,A -85,B 0,C 180,E1 -7752.335,E2 -7752.335} C_VEL
LIN {X 0,Y 469.2,Z 288.002,A -85,B 0,C 180,E1 -7753.266,E2 -7753.266} C_VEL
LIN {X 0,Y 469.606,Z 277.165,A -85,B 0,C 180,E1 -7753.965,E2 -7753.965} C_VEL
LIN {X 0,Y 470.059,Z 265.268,A -85,B 0,C 180,E1 -7754.559,E2 -7754.559} C_VEL
LIN {X 0,Y 470.005,Z 257.506,A -85,B 0,C 180,E1 -7754.865,E2 -7754.865} C_VEL
LIN {X 0,Y 467.354,Z 243.999,A -85,B 0,C 180,E1 -7755.342,E2 -7755.342} C_VEL
LIN {X 0,Y 467.473,Z 234.853,A -85,B 0,C 180,E1 -7758.71,E2 -7758.71} C_VEL
LIN {X 0,Y 467.644,Z 226.984,A -85,B 0,C 180,E1 -7761.615,E2 -7761.615} C_VEL
LIN {X 0,Y 467.784,Z 218.179,A -85,B 0,C 180,E1 -7764.877,E2 -7764.877} C_VEL
LIN {X 0,Y 467.933,Z 210.452,A -85,B 0,C 180,E1 -7767.749,E2 -7767.749} C_VEL
LIN {X 0,Y 468.109,Z 202.518,A -85,B 0,C 180,E1 -7770.695,E2 -7770.695} C_VEL
LIN {X 0,Y 468.284,Z 194.321,A -85,B 0,C 180,E1 -7773.731,E2 -7773.731} C_VEL
LIN {X 0,Y 468.124,Z 188.648,A -85,B 0,C 180,E1 -7775.839,E2 -7775.839} C_VEL
LIN {X 0,Y 467.601,Z 185.242,A -85,B 0,C 180,E1 -7777.194,E2 -7777.194} C_VEL
LIN {X 0,Y 467.576,Z 185.241,A -85,B 0,C 180,E1 -7780.265,E2 -7780.265} C_VEL
LIN {X 0,Y 467.553,Z 185.244,A -85,B 0,C 180,E1 -7783.745,E2 -7783.745} C_VEL
LIN {X 0,Y 467.556,Z 185.245,A -85,B 0,C 180,E1 -7786.255,E2 -7786.255} C_VEL
LIN {X 0,Y 467.584,Z 185.241,A -85,B 0,C 180,E1 -7788.723,E2 -7788.723} C_VEL
LIN {X 0,Y 467.547,Z 185.247,A -85,B 0,C 180,E1 -7791.953,E2 -7791.953} C_VEL
LIN {X 0,Y 467.556,Z 185.247,A -85,B 0,C 180,E1 -7795.166,E2 -7795.166} C_VEL
LIN {X 0,Y 467.564,Z 185.244,A -85,B 0,C 180,E1 -7798.257,E2 -7798.257} C_VEL
LIN {X 0,Y 467.359,Z 185.273,A -85,B 0,C 180,E1 -7801.235,E2 -7801.235} C_VEL
LIN {X 0,Y 467.342,Z 187.462,A -85,B 0,C 180,E1 -7803.182,E2 -7803.182} C_VEL
LIN {X 0,Y 467.245,Z 190.994,A -85,B 0,C 180,E1 -7806.038,E2 -7806.038} C_VEL
LIN {X 0,Y 467.177,Z 193.497,A -85,B 0,C 180,E1 -7808.057,E2 -7808.057} C_VEL
LIN {X 0,Y 466.494,Z 194.472,A -85,B 0,C 180,E1 -7808.766,E2 -7808.766} C_VEL
LIN {X 0,Y 463.64,Z 196.272,A -85,B 0,C 180,E1 -7809.914,E2 -7809.914} C_VEL
LIN {X 0,Y 461.221,Z 197.739,A -85,B 0,C 180,E1 -7810.839,E2 -7810.839} C_VEL
LIN {X 0,Y 460.162,Z 198.783,A -85,B 0,C 180,E1 -7811.555,E2 -7811.555} C_VEL
LIN {X 0,Y 460.064,Z 199.106,A -85,B 0,C 180,E1 -7811.799,E2 -7811.799} C_VEL
LIN {X 0,Y 460.045,Z 203.266,A -85,B 0,C 180,E1 -7814.946,E2 -7814.946} C_VEL
LIN {X 0,Y 460.102,Z 208.424,A -85,B 0,C 180,E1 -7818.545,E2 -7818.545} C_VEL
LIN {X 0,Y 460.026,Z 211.111,A -85,B 0,C 180,E1 -7820.269,E2 -7820.269} C_VEL
LIN {X 0,Y 462.328,Z 221.929,A -85,B 0,C 180,E1 -7820.759,E2 -7820.759} C_VEL
LIN {X 0,Y 462.174,Z 230.74,A -85,B 0,C 180,E1 -7821.272,E2 -7821.272} C_VEL
LIN {X 0,Y 462.08,Z 237.425,A -85,B 0,C 180,E1 -7821.788,E2 -7821.788} C_VEL
LIN {X 0,Y 461.799,Z 244.271,A -85,B 0,C 180,E1 -7822.456,E2 -7822.456} C_VEL
LIN {X 0,Y 461.666,Z 250.393,A -85,B 0,C 180,E1 -7823.223,E2 -7823.223} C_VEL
LIN {X 0,Y 461.408,Z 255.845,A -85,B 0,C 180,E1 -7824.098,E2 -7824.098} C_VEL
LIN {X 0,Y 461.033,Z 260.988,A -85,B 0,C 180,E1 -7825.189,E2 -7825.189} C_VEL
LIN {X 0,Y 460.821,Z 265.298,A -85,B 0,C 180,E1 -7826.501,E2 -7826.501} C_VEL
LIN {X 0,Y 460.557,Z 267.287,A -85,B 0,C 180,E1 -7827.375,E2 -7827.375} C_VEL
LIN {X 0,Y 460.542,Z 268.627,A -85,B 0,C 180,E1 -7828.25,E2 -7828.25} C_VEL
LIN {X 0,Y 460.451,Z 269.422,A -85,B 0,C 180,E1 -7829.124,E2 -7829.124} C_VEL
LIN {X 0,Y 460.416,Z 269.697,A -85,B 0,C 180,E1 -7829.999,E2 -7829.999} C_VEL
LIN {X 0,Y 460.443,Z 269.474,A -85,B 0,C 180,E1 -7830.873,E2 -7830.873} C_VEL
LIN {X 0,Y 460.501,Z 268.739,A -85,B 0,C 180,E1 -7831.748,E2 -7831.748} C_VEL
LIN {X 0,Y 460.55,Z 267.456,A -85,B 0,C 180,E1 -7832.623,E2 -7832.623} C_VEL
LIN {X 0,Y 460.946,Z 264.322,A -85,B 0,C 180,E1 -7833.933,E2 -7833.933} C_VEL
LIN {X 0,Y 461.067,Z 259.56,A -85,B 0,C 180,E1 -7835.246,E2 -7835.246} C_VEL
LIN {X 0,Y 461.372,Z 256.344,A -85,B 0,C 180,E1 -7835.9,E2 -7835.9} C_VEL
LIN {X 0,Y 461.635,Z 251.074,A -85,B 0,C 180,E1 -7836.775,E2 -7836.775} C_VEL
LIN {X 0,Y 461.837,Z 244.128,A -85,B 0,C 180,E1 -7837.651,E2 -7837.651} C_VEL
LIN {X 0,Y 462.053,Z 237.621,A -85,B 0,C 180,E1 -7838.289,E2 -7838.289} C_VEL
LIN {X 0,Y 462.239,Z 230.315,A -85,B 0,C 180,E1 -7838.854,E2 -7838.854} C_VEL
LIN {X 0,Y 462.281,Z 221.633,A -85,B 0,C 180,E1 -7839.35,E2 -7839.35} C_VEL
LIN {X 0,Y 460.032,Z 211.086,A -85,B 0,C 180,E1 -7839.84,E2 -7839.84} C_VEL
LIN {X 0,Y 460.061,Z 207.247,A -85,B 0,C 180,E1 -7842.348,E2 -7842.348} C_VEL
LIN {X 0,Y 460.073,Z 202.181,A -85,B 0,C 180,E1 -7845.959,E2 -7845.959} C_VEL
LIN {X 0,Y 460.108,Z 198.561,A -85,B 0,C 180,E1 -7848.731,E2 -7848.731} C_VEL
LIN {X 0,Y 460.133,Z 195.025,A -85,B 0,C 180,E1 -7851.503,E2 -7851.503} C_VEL
LIN {X 0,Y 460.188,Z 191.514,A -85,B 0,C 180,E1 -7854.351,E2 -7854.351} C_VEL
LIN {X 0,Y 460.312,Z 187.901,A -85,B 0,C 180,E1 -7857.259,E2 -7857.259} C_VEL
LIN {X 0,Y 460.283,Z 186.674,A -85,B 0,C 180,E1 -7858.249,E2 -7858.249} C_VEL
LIN {X 0,Y 460.389,Z 186.14,A -85,B 0,C 180,E1 -7859.526,E2 -7859.526} C_VEL
LIN {X 0,Y 460.525,Z 186.118,A -85,B 0,C 180,E1 -7862.283,E2 -7862.283} C_VEL
LIN {X 0,Y 460.508,Z 186.125,A -85,B 0,C 180,E1 -7865.444,E2 -7865.444} C_VEL
LIN {X 0,Y 460.539,Z 186.118,A -85,B 0,C 180,E1 -7868.896,E2 -7868.896} C_VEL
LIN {X 0,Y 460.518,Z 186.118,A -85,B 0,C 180,E1 -7872.18,E2 -7872.18} C_VEL
LIN {X 0,Y 460.51,Z 186.121,A -85,B 0,C 180,E1 -7875.41,E2 -7875.41} C_VEL
LIN {X 0,Y 460.525,Z 186.119,A -85,B 0,C 180,E1 -7878.396,E2 -7878.396} C_VEL
LIN {X 0,Y 460.523,Z 186.118,A -85,B 0,C 180,E1 -7881.266,E2 -7881.266} C_VEL
LIN {X 0,Y 460.505,Z 186.126,A -85,B 0,C 180,E1 -7884.554,E2 -7884.554} C_VEL
LIN {X 0,Y 460.524,Z 186.117,A -85,B 0,C 180,E1 -7887.715,E2 -7887.715} C_VEL
LIN {X 0,Y 460.538,Z 186.115,A -85,B 0,C 180,E1 -7890.769,E2 -7890.769} C_VEL
LIN {X 0,Y 460.558,Z 186.115,A -85,B 0,C 180,E1 -7893.734,E2 -7893.734} C_VEL
LIN {X 0,Y 460.536,Z 186.117,A -85,B 0,C 180,E1 -7896.623,E2 -7896.623} C_VEL
LIN {X 0,Y 460.542,Z 186.114,A -85,B 0,C 180,E1 -7899.452,E2 -7899.452} C_VEL
LIN {X 0,Y 460.549,Z 186.116,A -85,B 0,C 180,E1 -7902.23,E2 -7902.23} C_VEL
LIN {X 0,Y 460.558,Z 186.107,A -85,B 0,C 180,E1 -7904.965,E2 -7904.965} C_VEL
LIN {X 0,Y 460.602,Z 186.106,A -85,B 0,C 180,E1 -7908.559,E2 -7908.559} C_VEL
LIN {X 0,Y 460.684,Z 186.097,A -85,B 0,C 180,E1 -7912.108,E2 -7912.108} C_VEL
LIN {X 0,Y 460.682,Z 186.096,A -85,B 0,C 180,E1 -7914.748,E2 -7914.748} C_VEL
LIN {X 0,Y 460.812,Z 186.084,A -85,B 0,C 180,E1 -7917.378,E2 -7917.378} C_VEL
LIN {X 0,Y 460.839,Z 186.071,A -85,B 0,C 180,E1 -7920,E2 -7920} C_VEL
LIN {X 0,Y 460.786,Z 186.088,A -85,B 0,C 180,E1 -7922.623,E2 -7922.623} C_VEL
LIN {X 0,Y 460.687,Z 186.096,A -85,B 0,C 180,E1 -7926.13,E2 -7926.13} C_VEL
LIN {X 0,Y 460.614,Z 186.106,A -85,B 0,C 180,E1 -7928.776,E2 -7928.776} C_VEL
LIN {X 0,Y 460.584,Z 186.113,A -85,B 0,C 180,E1 -7932.436,E2 -7932.436} C_VEL
LIN {X 0,Y 460.588,Z 186.114,A -85,B 0,C 180,E1 -7935.998,E2 -7935.998} C_VEL
LIN {X 0,Y 460.555,Z 186.116,A -85,B 0,C 180,E1 -7939.616,E2 -7939.616} C_VEL
LIN {X 0,Y 460.495,Z 186.124,A -85,B 0,C 180,E1 -7942.43,E2 -7942.43} C_VEL
LIN {X 0,Y 460.522,Z 186.124,A -85,B 0,C 180,E1 -7945.794,E2 -7945.794} C_VEL
LIN {X 0,Y 460.507,Z 186.123,A -85,B 0,C 180,E1 -7949.233,E2 -7949.233} C_VEL
LIN {X 0,Y 460.519,Z 186.118,A -85,B 0,C 180,E1 -7952.285,E2 -7952.285} C_VEL
LIN {X 0,Y 460.496,Z 186.127,A -85,B 0,C 180,E1 -7955.447,E2 -7955.447} C_VEL
LIN {X 0,Y 460.519,Z 186.124,A -85,B 0,C 180,E1 -7958.896,E2 -7958.896} C_VEL
LIN {X 0,Y 460.494,Z 186.123,A -85,B 0,C 180,E1 -7962.185,E2 -7962.185} C_VEL
LIN {X 0,Y 460.506,Z 186.122,A -85,B 0,C 180,E1 -7965.412,E2 -7965.412} C_VEL
LIN {X 0,Y 460.525,Z 186.114,A -85,B 0,C 180,E1 -7968.399,E2 -7968.399} C_VEL
LIN {X 0,Y 460.52,Z 186.119,A -85,B 0,C 180,E1 -7971.268,E2 -7971.268} C_VEL
LIN {X 0,Y 460.552,Z 186.193,A -85,B 0,C 180,E1 -7974.794,E2 -7974.794} C_VEL
LIN {X 0,Y 463.286,Z 198.105,A -85,B 0,C 180,E1 -7977.675,E2 -7977.675} C_VEL
LIN {X 0,Y 465.049,Z 206.069,A -85,B 0,C 180,E1 -7979.475,E2 -7979.475} C_VEL
LIN {X 0,Y 464.863,Z 211.587,A -85,B 0,C 180,E1 -7980.572,E2 -7980.572} C_VEL
LIN {X 0,Y 463.582,Z 228.151,A -85,B 0,C 180,E1 -7983.725,E2 -7983.725} C_VEL
LIN {X 0,Y 462.484,Z 245.752,A -85,B 0,C 180,E1 -7986.966,E2 -7986.966} C_VEL
LIN {X 0,Y 461.62,Z 262.238,A -85,B 0,C 180,E1 -7989.969,E2 -7989.969} C_VEL
LIN {X 0,Y 460.791,Z 280.83,A -85,B 0,C 180,E1 -7993.407,E2 -7993.407} C_VEL
LIN {X 0,Y 460.581,Z 287.009,A -85,B 0,C 180,E1 -7994.57,E2 -7994.57} C_VEL
LIN {X 0,Y 462.085,Z 304.082,A -85,B 0,C 180,E1 -7995.017,E2 -7995.017} C_VEL
LIN {X 0,Y 462.523,Z 311.535,A -85,B 0,C 180,E1 -7995.285,E2 -7995.285} C_VEL
LIN {X 0,Y 462.16,Z 324.443,A -85,B 0,C 180,E1 -7995.863,E2 -7995.863} C_VEL
LIN {X 0,Y 461.675,Z 336.348,A -85,B 0,C 180,E1 -7996.578,E2 -7996.578} C_VEL
LIN {X 0,Y 461.232,Z 346.747,A -85,B 0,C 180,E1 -7997.374,E2 -7997.374} C_VEL
LIN {X 0,Y 460.792,Z 358.048,A -85,B 0,C 180,E1 -7998.454,E2 -7998.454} C_VEL
LIN {X 0,Y 460.445,Z 366.504,A -85,B 0,C 180,E1 -7999.447,E2 -7999.447} C_VEL
LIN {X 0,Y 460.127,Z 375.658,A -85,B 0,C 180,E1 -8000.772,E2 -8000.772} C_VEL
LIN {X 0,Y 459.895,Z 383.012,A -85,B 0,C 180,E1 -8002.096,E2 -8002.096} C_VEL
LIN {X 0,Y 459.744,Z 389.315,A -85,B 0,C 180,E1 -8003.536,E2 -8003.536} C_VEL
LIN {X 0,Y 459.786,Z 393.447,A -85,B 0,C 180,E1 -8004.739,E2 -8004.739} C_VEL
LIN {X 0,Y 459.722,Z 395.834,A -85,B 0,C 180,E1 -8005.617,E2 -8005.617} C_VEL
LIN {X 0,Y 459.781,Z 397.781,A -85,B 0,C 180,E1 -8006.496,E2 -8006.496} C_VEL
LIN {X 0,Y 459.738,Z 399.273,A -85,B 0,C 180,E1 -8007.373,E2 -8007.373} C_VEL
LIN {X 0,Y 459.726,Z 400.296,A -85,B 0,C 180,E1 -8008.249,E2 -8008.249} C_VEL
LIN {X 0,Y 459.695,Z 400.911,A -85,B 0,C 180,E1 -8009.125,E2 -8009.125} C_VEL
LIN {X 0,Y 459.701,Z 401.122,A -85,B 0,C 180,E1 -8010.001,E2 -8010.001} C_VEL
LIN {X 0,Y 459.697,Z 400.873,A -85,B 0,C 180,E1 -8010.877,E2 -8010.877} C_VEL
LIN {X 0,Y 459.732,Z 400.205,A -85,B 0,C 180,E1 -8011.753,E2 -8011.753} C_VEL
LIN {X 0,Y 459.743,Z 399.128,A -85,B 0,C 180,E1 -8012.63,E2 -8012.63} C_VEL
LIN {X 0,Y 459.756,Z 396.668,A -85,B 0,C 180,E1 -8013.946,E2 -8013.946} C_VEL
LIN {X 0,Y 459.793,Z 393.168,A -85,B 0,C 180,E1 -8015.263,E2 -8015.263} C_VEL
LIN {X 0,Y 459.801,Z 387.761,A -85,B 0,C 180,E1 -8016.774,E2 -8016.774} C_VEL
LIN {X 0,Y 459.936,Z 381.47,A -85,B 0,C 180,E1 -8018.127,E2 -8018.127} C_VEL
LIN {X 0,Y 460.176,Z 373.82,A -85,B 0,C 180,E1 -8019.451,E2 -8019.451} C_VEL
LIN {X 0,Y 460.418,Z 366.03,A -85,B 0,C 180,E1 -8020.556,E2 -8020.556} C_VEL
LIN {X 0,Y 460.842,Z 356.57,A -85,B 0,C 180,E1 -8021.659,E2 -8021.659} C_VEL
LIN {X 0,Y 461.244,Z 344.526,A -85,B 0,C 180,E1 -8022.793,E2 -8022.793} C_VEL
LIN {X 0,Y 461.86,Z 333.027,A -85,B 0,C 180,E1 -8023.643,E2 -8023.643} C_VEL
LIN {X 0,Y 462.41,Z 319.616,A -85,B 0,C 180,E1 -8024.412,E2 -8024.412} C_VEL
LIN {X 0,Y 462.651,Z 309.493,A -85,B 0,C 180,E1 -8024.854,E2 -8024.854} C_VEL
LIN {X 0,Y 461.825,Z 296.561,A -85,B 0,C 180,E1 -8025.305,E2 -8025.305} C_VEL
LIN {X 0,Y 460.609,Z 286.097,A -85,B 0,C 180,E1 -8025.601,E2 -8025.601} C_VEL
LIN {X 0,Y 461.29,Z 268.256,A -85,B 0,C 180,E1 -8028.925,E2 -8028.925} C_VEL
LIN {X 0,Y 462.168,Z 251.002,A -85,B 0,C 180,E1 -8032.078,E2 -8032.078} C_VEL
LIN {X 0,Y 463.155,Z 234.212,A -85,B 0,C 180,E1 -8035.144,E2 -8035.144} C_VEL
LIN {X 0,Y 464.363,Z 217.258,A -85,B 0,C 180,E1 -8038.322,E2 -8038.322} C_VEL
LIN {X 0,Y 465.143,Z 207.568,A -85,B 0,C 180,E1 -8040.21,E2 -8040.21} C_VEL
LIN {X 0,Y 464.12,Z 201.669,A -85,B 0,C 180,E1 -8041.496,E2 -8041.496} C_VEL
LIN {X 0,Y 461.126,Z 188.543,A -85,B 0,C 180,E1 -8044.612,E2 -8044.612} C_VEL
LIN {X 0,Y 460.537,Z 186.124,A -85,B 0,C 180,E1 -8045.268,E2 -8045.268} C_VEL
LIN {X 0,Y 460.536,Z 186.121,A -85,B 0,C 180,E1 -8048.896,E2 -8048.896} C_VEL
LIN {X 0,Y 460.528,Z 186.121,A -85,B 0,C 180,E1 -8052.182,E2 -8052.182} C_VEL
LIN {X 0,Y 460.519,Z 186.122,A -85,B 0,C 180,E1 -8055.411,E2 -8055.411} C_VEL
LIN {X 0,Y 460.537,Z 186.12,A -85,B 0,C 180,E1 -8058.398,E2 -8058.398} C_VEL
LIN {X 0,Y 460.52,Z 186.124,A -85,B 0,C 180,E1 -8061.266,E2 -8061.266} C_VEL
LIN {X 0,Y 460.506,Z 186.279,A -85,B 0,C 180,E1 -8063.337,E2 -8063.337} C_VEL
LIN {X 0,Y 461.611,Z 191.982,A -85,B 0,C 180,E1 -8065.301,E2 -8065.301} C_VEL
LIN {X 0,Y 461.555,Z 198.133,A -85,B 0,C 180,E1 -8067.328,E2 -8067.328} C_VEL
LIN {X 0,Y 461.294,Z 206.925,A -85,B 0,C 180,E1 -8070.277,E2 -8070.277} C_VEL
LIN {X 0,Y 461.18,Z 214.088,A -85,B 0,C 180,E1 -8072.795,E2 -8072.795} C_VEL
LIN {X 0,Y 461.088,Z 222.379,A -85,B 0,C 180,E1 -8075.698,E2 -8075.698} C_VEL
LIN {X 0,Y 460.91,Z 231.656,A -85,B 0,C 180,E1 -8079.002,E2 -8079.002} C_VEL
LIN {X 0,Y 460.708,Z 240.519,A -85,B 0,C 180,E1 -8082.236,E2 -8082.236} C_VEL
LIN {X 0,Y 460.625,Z 246.266,A -85,B 0,C 180,E1 -8084.344,E2 -8084.344} C_VEL
LIN {X 0,Y 463.413,Z 258.581,A -85,B 0,C 180,E1 -8084.848,E2 -8084.848} C_VEL
LIN {X 0,Y 463.637,Z 261.806,A -85,B 0,C 180,E1 -8084.982,E2 -8084.982} C_VEL
LIN {X 0,Y 463.25,Z 273.223,A -85,B 0,C 180,E1 -8085.503,E2 -8085.503} C_VEL
LIN {X 0,Y 462.801,Z 285.533,A -85,B 0,C 180,E1 -8086.251,E2 -8086.251} C_VEL
LIN {X 0,Y 462.276,Z 297.217,A -85,B 0,C 180,E1 -8087.153,E2 -8087.153} C_VEL
LIN {X 0,Y 461.684,Z 308.447,A -85,B 0,C 180,E1 -8088.252,E2 -8088.252} C_VEL
LIN {X 0,Y 461.14,Z 318.379,A -85,B 0,C 180,E1 -8089.462,E2 -8089.462} C_VEL
LIN {X 0,Y 460.76,Z 327.029,A -85,B 0,C 180,E1 -8090.784,E2 -8090.784} C_VEL
LIN {X 0,Y 460.356,Z 334.036,A -85,B 0,C 180,E1 -8092.103,E2 -8092.103} C_VEL
LIN {X 0,Y 460.137,Z 339.61,A -85,B 0,C 180,E1 -8093.423,E2 -8093.423} C_VEL
LIN {X 0,Y 459.803,Z 343.963,A -85,B 0,C 180,E1 -8094.738,E2 -8094.738} C_VEL
LIN {X 0,Y 459.904,Z 346.224,A -85,B 0,C 180,E1 -8095.618,E2 -8095.618} C_VEL
LIN {X 0,Y 459.797,Z 348.076,A -85,B 0,C 180,E1 -8096.495,E2 -8096.495} C_VEL
LIN {X 0,Y 459.776,Z 349.487,A -85,B 0,C 180,E1 -8097.372,E2 -8097.372} C_VEL
LIN {X 0,Y 459.564,Z 351.047,A -85,B 0,C 180,E1 -8099.124,E2 -8099.124} C_VEL
LIN {X 0,Y 459.544,Z 351.236,A -85,B 0,C 180,E1 -8100,E2 -8100} C_VEL
LIN {X 0,Y 459.562,Z 350.98,A -85,B 0,C 180,E1 -8100.876,E2 -8100.876} C_VEL
LIN {X 0,Y 459.64,Z 350.323,A -85,B 0,C 180,E1 -8101.752,E2 -8101.752} C_VEL
LIN {X 0,Y 459.716,Z 349.275,A -85,B 0,C 180,E1 -8102.629,E2 -8102.629} C_VEL
LIN {X 0,Y 459.782,Z 347.802,A -85,B 0,C 180,E1 -8103.505,E2 -8103.505} C_VEL
LIN {X 0,Y 459.78,Z 344.77,A -85,B 0,C 180,E1 -8104.823,E2 -8104.823} C_VEL
LIN {X 0,Y 460.003,Z 340.666,A -85,B 0,C 180,E1 -8106.139,E2 -8106.139} C_VEL
LIN {X 0,Y 460.165,Z 334.383,A -85,B 0,C 180,E1 -8107.68,E2 -8107.68} C_VEL
LIN {X 0,Y 460.526,Z 327.539,A -85,B 0,C 180,E1 -8108.999,E2 -8108.999} C_VEL
LIN {X 0,Y 460.895,Z 318.963,A -85,B 0,C 180,E1 -8110.322,E2 -8110.322} C_VEL
LIN {X 0,Y 461.331,Z 310.207,A -85,B 0,C 180,E1 -8111.423,E2 -8111.423} C_VEL
LIN {X 0,Y 461.842,Z 299.587,A -85,B 0,C 180,E1 -8112.513,E2 -8112.513} C_VEL
LIN {X 0,Y 462.291,Z 287.253,A -85,B 0,C 180,E1 -8113.517,E2 -8113.517} C_VEL
LIN {X 0,Y 462.802,Z 275.007,A -85,B 0,C 180,E1 -8114.286,E2 -8114.286} C_VEL
LIN {X 0,Y 463.21,Z 262.222,A -85,B 0,C 180,E1 -8114.891,E2 -8114.891} C_VEL
LIN {X 0,Y 463.065,Z 258.436,A -85,B 0,C 180,E1 -8115.042,E2 -8115.042} C_VEL
LIN {X 0,Y 460.473,Z 245.347,A -85,B 0,C 180,E1 -8115.516,E2 -8115.516} C_VEL
LIN {X 0,Y 460.287,Z 244.284,A -85,B 0,C 180,E1 -8115.561,E2 -8115.561} C_VEL
LIN {X 0,Y 460.426,Z 235.815,A -85,B 0,C 180,E1 -8118.696,E2 -8118.696} C_VEL
LIN {X 0,Y 460.6,Z 228.31,A -85,B 0,C 180,E1 -8121.482,E2 -8121.482} C_VEL
LIN {X 0,Y 460.763,Z 219.411,A -85,B 0,C 180,E1 -8124.8,E2 -8124.8} C_VEL
LIN {X 0,Y 460.939,Z 210.286,A -85,B 0,C 180,E1 -8128.207,E2 -8128.207} C_VEL
LIN {X 0,Y 461.104,Z 203.6,A -85,B 0,C 180,E1 -8130.704,E2 -8130.704} C_VEL
LIN {X 0,Y 461.277,Z 195.337,A -85,B 0,C 180,E1 -8133.788,E2 -8133.788} C_VEL
LIN {X 0,Y 461.245,Z 191.085,A -85,B 0,C 180,E1 -8135.381,E2 -8135.381} C_VEL
LIN {X 0,Y 460.55,Z 186.12,A -85,B 0,C 180,E1 -8137.325,E2 -8137.325} C_VEL
LIN {X 0,Y 460.54,Z 186.118,A -85,B 0,C 180,E1 -8140.268,E2 -8140.268} C_VEL
LIN {X 0,Y 460.514,Z 186.121,A -85,B 0,C 180,E1 -8143.374,E2 -8143.374} C_VEL
LIN {X 0,Y 460.502,Z 186.122,A -85,B 0,C 180,E1 -8146.624,E2 -8146.624} C_VEL
LIN {X 0,Y 460.543,Z 186.118,A -85,B 0,C 180,E1 -8149.731,E2 -8149.731} C_VEL
LIN {X 0,Y 460.486,Z 186.129,A -85,B 0,C 180,E1 -8152.527,E2 -8152.527} C_VEL
LIN {X 0,Y 460.539,Z 186.123,A -85,B 0,C 180,E1 -8155.622,E2 -8155.622} C_VEL
LIN {X 0,Y 460.509,Z 186.126,A -85,B 0,C 180,E1 -8158.741,E2 -8158.741} C_VEL
LIN {X 0,Y 460.387,Z 186.141,A -85,B 0,C 180,E1 -8160.757,E2 -8160.757} C_VEL
LIN {X 0,Y 460.289,Z 186.569,A -85,B 0,C 180,E1 -8161.748,E2 -8161.748} C_VEL
LIN {X 0,Y 460.28,Z 190.195,A -85,B 0,C 180,E1 -8164.688,E2 -8164.688} C_VEL
LIN {X 0,Y 460.143,Z 193.735,A -85,B 0,C 180,E1 -8167.551,E2 -8167.551} C_VEL
LIN {X 0,Y 460.077,Z 197.244,A -85,B 0,C 180,E1 -8170.362,E2 -8170.362} C_VEL
LIN {X 0,Y 460.064,Z 199.106,A -85,B 0,C 180,E1 -8171.799,E2 -8171.799} C_VEL
LIN {X 0,Y 459.361,Z 200.132,A -85,B 0,C 180,E1 -8172.518,E2 -8172.518} C_VEL
LIN {X 0,Y 456.479,Z 202.031,A -85,B 0,C 180,E1 -8173.682,E2 -8173.682} C_VEL
LIN {X 0,Y 454.071,Z 203.59,A -85,B 0,C 180,E1 -8174.62,E2 -8174.62} C_VEL
LIN {X 0,Y 453.054,Z 204.708,A -85,B 0,C 180,E1 -8175.347,E2 -8175.347} C_VEL
LIN {X 0,Y 452.979,Z 205.059,A -85,B 0,C 180,E1 -8175.593,E2 -8175.593} C_VEL
LIN {X 0,Y 453.078,Z 209.06,A -85,B 0,C 180,E1 -8178.365,E2 -8178.365} C_VEL
LIN {X 0,Y 452.98,Z 211.697,A -85,B 0,C 180,E1 -8180.06,E2 -8180.06} C_VEL
LIN {X 0,Y 455.326,Z 222.398,A -85,B 0,C 180,E1 -8180.56,E2 -8180.56} C_VEL
LIN {X 0,Y 455.306,Z 230.206,A -85,B 0,C 180,E1 -8181.007,E2 -8181.007} C_VEL
LIN {X 0,Y 455.157,Z 238.408,A -85,B 0,C 180,E1 -8181.64,E2 -8181.64} C_VEL
LIN {X 0,Y 454.858,Z 245.437,A -85,B 0,C 180,E1 -8182.341,E2 -8182.341} C_VEL
LIN {X 0,Y 454.705,Z 251.502,A -85,B 0,C 180,E1 -8183.119,E2 -8183.119} C_VEL
LIN {X 0,Y 454.429,Z 256.898,A -85,B 0,C 180,E1 -8184.007,E2 -8184.007} C_VEL
LIN {X 0,Y 454.04,Z 262.013,A -85,B 0,C 180,E1 -8185.115,E2 -8185.115} C_VEL
LIN {X 0,Y 453.82,Z 266.294,A -85,B 0,C 180,E1 -8186.447,E2 -8186.447} C_VEL
LIN {X 0,Y 453.543,Z 268.274,A -85,B 0,C 180,E1 -8187.334,E2 -8187.334} C_VEL
LIN {X 0,Y 453.526,Z 269.606,A -85,B 0,C 180,E1 -8188.223,E2 -8188.223} C_VEL
LIN {X 0,Y 453.431,Z 270.397,A -85,B 0,C 180,E1 -8189.111,E2 -8189.111} C_VEL
LIN {X 0,Y 453.394,Z 270.671,A -85,B 0,C 180,E1 -8189.999,E2 -8189.999} C_VEL
LIN {X 0,Y 453.423,Z 270.447,A -85,B 0,C 180,E1 -8190.887,E2 -8190.887} C_VEL
LIN {X 0,Y 453.489,Z 269.715,A -85,B 0,C 180,E1 -8191.775,E2 -8191.775} C_VEL
LIN {X 0,Y 453.536,Z 268.439,A -85,B 0,C 180,E1 -8192.663,E2 -8192.663} C_VEL
LIN {X 0,Y 453.956,Z 265.319,A -85,B 0,C 180,E1 -8193.994,E2 -8193.994} C_VEL
LIN {X 0,Y 454.073,Z 260.588,A -85,B 0,C 180,E1 -8195.327,E2 -8195.327} C_VEL
LIN {X 0,Y 454.392,Z 257.392,A -85,B 0,C 180,E1 -8195.991,E2 -8195.991} C_VEL
LIN {X 0,Y 454.631,Z 250.582,A -85,B 0,C 180,E1 -8197.103,E2 -8197.103} C_VEL
LIN {X 0,Y 454.934,Z 244.268,A -85,B 0,C 180,E1 -8197.879,E2 -8197.879} C_VEL
LIN {X 0,Y 455.168,Z 236.824,A -85,B 0,C 180,E1 -8198.595,E2 -8198.595} C_VEL
LIN {X 0,Y 455.366,Z 228.236,A -85,B 0,C 180,E1 -8199.213,E2 -8199.213} C_VEL
LIN {X 0,Y 455.251,Z 222.077,A -85,B 0,C 180,E1 -8199.551,E2 -8199.551} C_VEL
LIN {X 0,Y 452.98,Z 211.719,A -85,B 0,C 180,E1 -8200.023,E2 -8200.023} C_VEL
LIN {X 0,Y 453.006,Z 207.865,A -85,B 0,C 180,E1 -8202.543,E2 -8202.543} C_VEL
LIN {X 0,Y 453.032,Z 202.725,A -85,B 0,C 180,E1 -8206.213,E2 -8206.213} C_VEL
LIN {X 0,Y 453.043,Z 199.082,A -85,B 0,C 180,E1 -8209.011,E2 -8209.011} C_VEL
LIN {X 0,Y 453.097,Z 195.465,A -85,B 0,C 180,E1 -8211.854,E2 -8211.854} C_VEL
LIN {X 0,Y 453.184,Z 191.901,A -85,B 0,C 180,E1 -8214.752,E2 -8214.752} C_VEL
LIN {X 0,Y 453.275,Z 188.237,A -85,B 0,C 180,E1 -8217.718,E2 -8217.718} C_VEL
LIN {X 0,Y 453.238,Z 187.032,A -85,B 0,C 180,E1 -8218.729,E2 -8218.729} C_VEL
LIN {X 0,Y 453.461,Z 187.002,A -85,B 0,C 180,E1 -8221.523,E2 -8221.523} C_VEL
LIN {X 0,Y 453.484,Z 186.996,A -85,B 0,C 180,E1 -8224.776,E2 -8224.776} C_VEL
LIN {X 0,Y 453.468,Z 186.997,A -85,B 0,C 180,E1 -8228.309,E2 -8228.309} C_VEL
LIN {X 0,Y 453.488,Z 186.995,A -85,B 0,C 180,E1 -8230.608,E2 -8230.608} C_VEL
LIN {X 0,Y 453.457,Z 187.001,A -85,B 0,C 180,E1 -8233.244,E2 -8233.244} C_VEL
LIN {X 0,Y 453.459,Z 186.997,A -85,B 0,C 180,E1 -8235.778,E2 -8235.778} C_VEL
LIN {X 0,Y 453.472,Z 186.997,A -85,B 0,C 180,E1 -8238.208,E2 -8238.208} C_VEL
LIN {X 0,Y 453.512,Z 186.997,A -85,B 0,C 180,E1 -8240.788,E2 -8240.788} C_VEL
LIN {X 0,Y 453.449,Z 186.998,A -85,B 0,C 180,E1 -8243.916,E2 -8243.916} C_VEL
LIN {X 0,Y 453.474,Z 186.995,A -85,B 0,C 180,E1 -8247.15,E2 -8247.15} C_VEL
LIN {X 0,Y 453.505,Z 186.993,A -85,B 0,C 180,E1 -8250.27,E2 -8250.27} C_VEL
LIN {X 0,Y 453.504,Z 186.991,A -85,B 0,C 180,E1 -8253.294,E2 -8253.294} C_VEL
LIN {X 0,Y 453.494,Z 186.998,A -85,B 0,C 180,E1 -8256.238,E2 -8256.238} C_VEL
LIN {X 0,Y 453.472,Z 186.993,A -85,B 0,C 180,E1 -8259.117,E2 -8259.117} C_VEL
LIN {X 0,Y 453.502,Z 186.997,A -85,B 0,C 180,E1 -8261.944,E2 -8261.944} C_VEL
LIN {X 0,Y 453.539,Z 186.981,A -85,B 0,C 180,E1 -8264.726,E2 -8264.726} C_VEL
LIN {X 0,Y 453.551,Z 186.984,A -85,B 0,C 180,E1 -8268.379,E2 -8268.379} C_VEL
LIN {X 0,Y 453.64,Z 186.975,A -85,B 0,C 180,E1 -8271.985,E2 -8271.985} C_VEL
LIN {X 0,Y 453.655,Z 186.971,A -85,B 0,C 180,E1 -8274.666,E2 -8274.666} C_VEL
LIN {X 0,Y 453.752,Z 186.964,A -85,B 0,C 180,E1 -8277.337,E2 -8277.337} C_VEL
LIN {X 0,Y 453.81,Z 186.947,A -85,B 0,C 180,E1 -8280,E2 -8280} C_VEL
LIN {X 0,Y 453.73,Z 186.968,A -85,B 0,C 180,E1 -8282.663,E2 -8282.663} C_VEL
LIN {X 0,Y 453.655,Z 186.973,A -85,B 0,C 180,E1 -8286.226,E2 -8286.226} C_VEL
LIN {X 0,Y 453.578,Z 186.981,A -85,B 0,C 180,E1 -8288.914,E2 -8288.914} C_VEL
LIN {X 0,Y 453.552,Z 186.987,A -85,B 0,C 180,E1 -8292.529,E2 -8292.529} C_VEL
LIN {X 0,Y 453.532,Z 186.994,A -85,B 0,C 180,E1 -8296.196,E2 -8296.196} C_VEL
LIN {X 0,Y 453.504,Z 186.992,A -85,B 0,C 180,E1 -8299.04,E2 -8299.04} C_VEL
LIN {X 0,Y 453.464,Z 187.003,A -85,B 0,C 180,E1 -8301.837,E2 -8301.837} C_VEL
LIN {X 0,Y 453.457,Z 186.999,A -85,B 0,C 180,E1 -8304.738,E2 -8304.738} C_VEL
LIN {X 0,Y 453.45,Z 187.004,A -85,B 0,C 180,E1 -8307.943,E2 -8307.943} C_VEL
LIN {X 0,Y 453.463,Z 186.998,A -85,B 0,C 180,E1 -8310.761,E2 -8310.761} C_VEL
LIN {X 0,Y 453.458,Z 186.997,A -85,B 0,C 180,E1 -8313.914,E2 -8313.914} C_VEL
LIN {X 0,Y 453.439,Z 187.004,A -85,B 0,C 180,E1 -8317.191,E2 -8317.191} C_VEL
LIN {X 0,Y 453.461,Z 186.993,A -85,B 0,C 180,E1 -8320.613,E2 -8320.613} C_VEL
LIN {X 0,Y 453.452,Z 186.999,A -85,B 0,C 180,E1 -8324.223,E2 -8324.223} C_VEL
LIN {X 0,Y 453.456,Z 186.998,A -85,B 0,C 180,E1 -8327.006,E2 -8327.006} C_VEL
LIN {X 0,Y 453.488,Z 186.998,A -85,B 0,C 180,E1 -8329.41,E2 -8329.41} C_VEL
LIN {X 0,Y 453.444,Z 187.005,A -85,B 0,C 180,E1 -8332.228,E2 -8332.228} C_VEL
LIN {X 0,Y 453.5,Z 187.121,A -85,B 0,C 180,E1 -8334.402,E2 -8334.402} C_VEL
LIN {X 0,Y 456.316,Z 199.135,A -85,B 0,C 180,E1 -8337.382,E2 -8337.382} C_VEL
LIN {X 0,Y 458.082,Z 207.102,A -85,B 0,C 180,E1 -8339.223,E2 -8339.223} C_VEL
LIN {X 0,Y 458.186,Z 211.313,A -85,B 0,C 180,E1 -8340.1,E2 -8340.1} C_VEL
LIN {X 0,Y 456.694,Z 228.775,A -85,B 0,C 180,E1 -8343.496,E2 -8343.496} C_VEL
LIN {X 0,Y 455.581,Z 245.223,A -85,B 0,C 180,E1 -8346.596,E2 -8346.596} C_VEL
LIN {X 0,Y 454.595,Z 262.845,A -85,B 0,C 180,E1 -8349.882,E2 -8349.882} C_VEL
LIN {X 0,Y 453.726,Z 281.138,A -85,B 0,C 180,E1 -8353.349,E2 -8353.349} C_VEL
LIN {X 0,Y 453.537,Z 286.295,A -85,B 0,C 180,E1 -8354.344,E2 -8354.344} C_VEL
LIN {X 0,Y 455.056,Z 302.794,A -85,B 0,C 180,E1 -8354.78,E2 -8354.78} C_VEL
LIN {X 0,Y 455.555,Z 312.63,A -85,B 0,C 180,E1 -8355.14,E2 -8355.14} C_VEL
LIN {X 0,Y 455.18,Z 325.651,A -85,B 0,C 180,E1 -8355.756,E2 -8355.756} C_VEL
LIN {X 0,Y 454.657,Z 337.122,A -85,B 0,C 180,E1 -8356.48,E2 -8356.48} C_VEL
LIN {X 0,Y 454.17,Z 348.345,A -85,B 0,C 180,E1 -8357.381,E2 -8357.381} C_VEL
LIN {X 0,Y 453.722,Z 358.422,A -85,B 0,C 180,E1 -8358.384,E2 -8358.384} C_VEL
LIN {X 0,Y 453.33,Z 367.558,A -85,B 0,C 180,E1 -8359.506,E2 -8359.506} C_VEL
LIN {X 0,Y 453.03,Z 376.471,A -85,B 0,C 180,E1 -8360.852,E2 -8360.852} C_VEL
LIN {X 0,Y 452.787,Z 383.578,A -85,B 0,C 180,E1 -8362.196,E2 -8362.196} C_VEL
LIN {X 0,Y 452.649,Z 389.303,A -85,B 0,C 180,E1 -8363.561,E2 -8363.561} C_VEL
LIN {X 0,Y 452.664,Z 394.252,A -85,B 0,C 180,E1 -8365.103,E2 -8365.103} C_VEL
LIN {X 0,Y 452.691,Z 397.353,A -85,B 0,C 180,E1 -8366.441,E2 -8366.441} C_VEL
LIN {X 0,Y 452.656,Z 398.86,A -85,B 0,C 180,E1 -8367.331,E2 -8367.331} C_VEL
LIN {X 0,Y 452.659,Z 399.893,A -85,B 0,C 180,E1 -8368.222,E2 -8368.222} C_VEL
LIN {X 0,Y 452.623,Z 400.513,A -85,B 0,C 180,E1 -8369.111,E2 -8369.111} C_VEL
LIN {X 0,Y 452.625,Z 400.729,A -85,B 0,C 180,E1 -8370.001,E2 -8370.001} C_VEL
LIN {X 0,Y 452.624,Z 400.491,A -85,B 0,C 180,E1 -8370.891,E2 -8370.891} C_VEL
LIN {X 0,Y 452.665,Z 399.824,A -85,B 0,C 180,E1 -8371.781,E2 -8371.781} C_VEL
LIN {X 0,Y 452.661,Z 398.746,A -85,B 0,C 180,E1 -8372.671,E2 -8372.671} C_VEL
LIN {X 0,Y 452.654,Z 396.287,A -85,B 0,C 180,E1 -8374.008,E2 -8374.008} C_VEL
LIN {X 0,Y 452.697,Z 392.793,A -85,B 0,C 180,E1 -8375.346,E2 -8375.346} C_VEL
LIN {X 0,Y 452.733,Z 387.687,A -85,B 0,C 180,E1 -8376.811,E2 -8376.811} C_VEL
LIN {X 0,Y 452.862,Z 381.119,A -85,B 0,C 180,E1 -8378.254,E2 -8378.254} C_VEL
LIN {X 0,Y 453.129,Z 373.479,A -85,B 0,C 180,E1 -8379.599,E2 -8379.599} C_VEL
LIN {X 0,Y 453.406,Z 365.719,A -85,B 0,C 180,E1 -8380.721,E2 -8380.721} C_VEL
LIN {X 0,Y 453.85,Z 356.321,A -85,B 0,C 180,E1 -8381.841,E2 -8381.841} C_VEL
LIN {X 0,Y 454.246,Z 345.288,A -85,B 0,C 180,E1 -8382.909,E2 -8382.909} C_VEL
LIN {X 0,Y 454.87,Z 334.609,A -85,B 0,C 180,E1 -8383.743,E2 -8383.743} C_VEL
LIN {X 0,Y 455.463,Z 321.898,A -85,B 0,C 180,E1 -8384.523,E2 -8384.523} C_VEL
LIN {X 0,Y 455.789,Z 309.954,A -85,B 0,C 180,E1 -8385.083,E2 -8385.083} C_VEL
LIN {X 0,Y 454.926,Z 296.233,A -85,B 0,C 180,E1 -8385.586,E2 -8385.586} C_VEL
LIN {X 0,Y 453.578,Z 284.817,A -85,B 0,C 180,E1 -8385.939,E2 -8385.939} C_VEL
LIN {X 0,Y 454.434,Z 265.831,A -85,B 0,C 180,E1 -8389.553,E2 -8389.553} C_VEL
LIN {X 0,Y 455.351,Z 248.986,A -85,B 0,C 180,E1 -8392.698,E2 -8392.698} C_VEL
LIN {X 0,Y 456.306,Z 233.768,A -85,B 0,C 180,E1 -8395.548,E2 -8395.548} C_VEL
LIN {X 0,Y 457.471,Z 218.666,A -85,B 0,C 180,E1 -8398.441,E2 -8398.441} C_VEL
LIN {X 0,Y 458.265,Z 208.788,A -85,B 0,C 180,E1 -8400.405,E2 -8400.405} C_VEL
LIN {X 0,Y 456.71,Z 200.924,A -85,B 0,C 180,E1 -8402.182,E2 -8402.182} C_VEL
LIN {X 0,Y 453.859,Z 188.56,A -85,B 0,C 180,E1 -8405.228,E2 -8405.228} C_VEL
LIN {X 0,Y 453.495,Z 187.001,A -85,B 0,C 180,E1 -8405.669,E2 -8405.669} C_VEL
LIN {X 0,Y 453.475,Z 186.999,A -85,B 0,C 180,E1 -8409.203,E2 -8409.203} C_VEL
LIN {X 0,Y 453.482,Z 187,A -85,B 0,C 180,E1 -8411.935,E2 -8411.935} C_VEL
LIN {X 0,Y 453.489,Z 186.998,A -85,B 0,C 180,E1 -8415.472,E2 -8415.472} C_VEL
LIN {X 0,Y 453.484,Z 186.999,A -85,B 0,C 180,E1 -8418.21,E2 -8418.21} C_VEL
LIN {X 0,Y 453.474,Z 187.003,A -85,B 0,C 180,E1 -8420.798,E2 -8420.798} C_VEL
LIN {X 0,Y 453.473,Z 187.03,A -85,B 0,C 180,E1 -8422.812,E2 -8422.812} C_VEL
LIN {X 0,Y 454.746,Z 193.518,A -85,B 0,C 180,E1 -8425.122,E2 -8425.122} C_VEL
LIN {X 0,Y 454.707,Z 199.832,A -85,B 0,C 180,E1 -8427.251,E2 -8427.251} C_VEL
LIN {X 0,Y 454.41,Z 208.942,A -85,B 0,C 180,E1 -8430.336,E2 -8430.336} C_VEL
LIN {X 0,Y 454.25,Z 217.369,A -85,B 0,C 180,E1 -8433.341,E2 -8433.341} C_VEL
LIN {X 0,Y 454.073,Z 226.89,A -85,B 0,C 180,E1 -8436.754,E2 -8436.754} C_VEL
LIN {X 0,Y 453.886,Z 236.014,A -85,B 0,C 180,E1 -8440.084,E2 -8440.084} C_VEL
LIN {X 0,Y 453.69,Z 244.861,A -85,B 0,C 180,E1 -8443.347,E2 -8443.347} C_VEL
LIN {X 0,Y 453.643,Z 246.728,A -85,B 0,C 180,E1 -8444.037,E2 -8444.037} C_VEL
LIN {X 0,Y 456.668,Z 259.692,A -85,B 0,C 180,E1 -8444.603,E2 -8444.603} C_VEL
LIN {X 0,Y 456.839,Z 264.026,A -85,B 0,C 180,E1 -8444.788,E2 -8444.788} C_VEL
LIN {X 0,Y 456.36,Z 276.271,A -85,B 0,C 180,E1 -8445.394,E2 -8445.394} C_VEL
LIN {X 0,Y 455.88,Z 288.102,A -85,B 0,C 180,E1 -8446.158,E2 -8446.158} C_VEL
LIN {X 0,Y 455.326,Z 299.183,A -85,B 0,C 180,E1 -8447.067,E2 -8447.067} C_VEL
LIN {X 0,Y 454.717,Z 310.124,A -85,B 0,C 180,E1 -8448.183,E2 -8448.183} C_VEL
LIN {X 0,Y 454.189,Z 318.971,A -85,B 0,C 180,E1 -8449.299,E2 -8449.299} C_VEL
LIN {X 0,Y 453.787,Z 327.59,A -85,B 0,C 180,E1 -8450.641,E2 -8450.641} C_VEL
LIN {X 0,Y 453.338,Z 334.564,A -85,B 0,C 180,E1 -8451.98,E2 -8451.98} C_VEL
LIN {X 0,Y 453.094,Z 340.344,A -85,B 0,C 180,E1 -8453.39,E2 -8453.39} C_VEL
LIN {X 0,Y 452.748,Z 344.433,A -85,B 0,C 180,E1 -8454.656,E2 -8454.656} C_VEL
LIN {X 0,Y 452.852,Z 346.686,A -85,B 0,C 180,E1 -8455.55,E2 -8455.55} C_VEL
LIN {X 0,Y 452.735,Z 348.53,A -85,B 0,C 180,E1 -8456.44,E2 -8456.44} C_VEL
LIN {X 0,Y 452.705,Z 349.923,A -85,B 0,C 180,E1 -8457.331,E2 -8457.331} C_VEL
LIN {X 0,Y 452.499,Z 351.458,A -85,B 0,C 180,E1 -8459.11,E2 -8459.11} C_VEL
LIN {X 0,Y 452.477,Z 351.631,A -85,B 0,C 180,E1 -8460,E2 -8460} C_VEL
LIN {X 0,Y 452.498,Z 351.357,A -85,B 0,C 180,E1 -8460.89,E2 -8460.89} C_VEL
LIN {X 0,Y 452.564,Z 350.686,A -85,B 0,C 180,E1 -8461.78,E2 -8461.78} C_VEL
LIN {X 0,Y 452.636,Z 349.623,A -85,B 0,C 180,E1 -8462.67,E2 -8462.67} C_VEL
LIN {X 0,Y 452.716,Z 348.124,A -85,B 0,C 180,E1 -8463.56,E2 -8463.56} C_VEL
LIN {X 0,Y 452.694,Z 345.061,A -85,B 0,C 180,E1 -8464.898,E2 -8464.898} C_VEL
LIN {X 0,Y 452.946,Z 340.92,A -85,B 0,C 180,E1 -8466.235,E2 -8466.235} C_VEL
LIN {X 0,Y 453.114,Z 334.594,A -85,B 0,C 180,E1 -8467.8,E2 -8467.8} C_VEL
LIN {X 0,Y 453.502,Z 327.701,A -85,B 0,C 180,E1 -8469.14,E2 -8469.14} C_VEL
LIN {X 0,Y 453.905,Z 319.061,A -85,B 0,C 180,E1 -8470.482,E2 -8470.482} C_VEL
LIN {X 0,Y 454.377,Z 310.25,A -85,B 0,C 180,E1 -8471.6,E2 -8471.6} C_VEL
LIN {X 0,Y 454.882,Z 299.706,A -85,B 0,C 180,E1 -8472.692,E2 -8472.692} C_VEL
LIN {X 0,Y 455.317,Z 288.623,A -85,B 0,C 180,E1 -8473.614,E2 -8473.614} C_VEL
LIN {X 0,Y 455.811,Z 276.759,A -85,B 0,C 180,E1 -8474.396,E2 -8474.396} C_VEL
LIN {X 0,Y 456.286,Z 264.467,A -85,B 0,C 180,E1 -8475.008,E2 -8475.008} C_VEL
LIN {X 0,Y 456.181,Z 259.564,A -85,B 0,C 180,E1 -8475.213,E2 -8475.213} C_VEL
LIN {X 0,Y 453.436,Z 245.628,A -85,B 0,C 180,E1 -8475.731,E2 -8475.731} C_VEL
LIN {X 0,Y 453.272,Z 244.605,A -85,B 0,C 180,E1 -8475.77,E2 -8475.77} C_VEL
LIN {X 0,Y 453.432,Z 235.91,A -85,B 0,C 180,E1 -8479.006,E2 -8479.006} C_VEL
LIN {X 0,Y 453.621,Z 227.079,A -85,B 0,C 180,E1 -8482.308,E2 -8482.308} C_VEL
LIN {X 0,Y 453.773,Z 218.034,A -85,B 0,C 180,E1 -8485.7,E2 -8485.7} C_VEL
LIN {X 0,Y 453.98,Z 210.123,A -85,B 0,C 180,E1 -8488.679,E2 -8488.679} C_VEL
LIN {X 0,Y 454.166,Z 201.947,A -85,B 0,C 180,E1 -8491.745,E2 -8491.745} C_VEL
LIN {X 0,Y 454.277,Z 193.514,A -85,B 0,C 180,E1 -8494.919,E2 -8494.919} C_VEL
LIN {X 0,Y 453.813,Z 188.788,A -85,B 0,C 180,E1 -8496.73,E2 -8496.73} C_VEL
LIN {X 0,Y 453.52,Z 186.995,A -85,B 0,C 180,E1 -8497.479,E2 -8497.479} C_VEL
LIN {X 0,Y 453.499,Z 186.996,A -85,B 0,C 180,E1 -8500.609,E2 -8500.609} C_VEL
LIN {X 0,Y 453.465,Z 187.003,A -85,B 0,C 180,E1 -8504.221,E2 -8504.221} C_VEL
LIN {X 0,Y 453.467,Z 186.999,A -85,B 0,C 180,E1 -8507.004,E2 -8507.004} C_VEL
LIN {X 0,Y 453.5,Z 186.997,A -85,B 0,C 180,E1 -8509.409,E2 -8509.409} C_VEL
LIN {X 0,Y 453.441,Z 187.005,A -85,B 0,C 180,E1 -8512.808,E2 -8512.808} C_VEL
LIN {X 0,Y 453.471,Z 187,A -85,B 0,C 180,E1 -8516.086,E2 -8516.086} C_VEL
LIN {X 0,Y 453.437,Z 187.005,A -85,B 0,C 180,E1 -8519.237,E2 -8519.237} C_VEL
LIN {X 0,Y 453.267,Z 187.028,A -85,B 0,C 180,E1 -8521.27,E2 -8521.27} C_VEL
LIN {X 0,Y 453.276,Z 190.551,A -85,B 0,C 180,E1 -8524.269,E2 -8524.269} C_VEL
LIN {X 0,Y 453.132,Z 194.163,A -85,B 0,C 180,E1 -8527.185,E2 -8527.185} C_VEL
LIN {X 0,Y 453.03,Z 197.719,A -85,B 0,C 180,E1 -8530.043,E2 -8530.043} C_VEL
LIN {X 0,Y 452.999,Z 201.365,A -85,B 0,C 180,E1 -8532.855,E2 -8532.855} C_VEL
LIN {X 0,Y 452.979,Z 205.059,A -85,B 0,C 180,E1 -8535.593,E2 -8535.593} C_VEL
LIN {X 0,Y 452.328,Z 206.173,A -85,B 0,C 180,E1 -8536.323,E2 -8536.323} C_VEL
LIN {X 0,Y 449.469,Z 208.256,A -85,B 0,C 180,E1 -8537.501,E2 -8537.501} C_VEL
LIN {X 0,Y 447.048,Z 209.987,A -85,B 0,C 180,E1 -8538.451,E2 -8538.451} C_VEL
LIN {X 0,Y 446.021,Z 211.245,A -85,B 0,C 180,E1 -8539.186,E2 -8539.186} C_VEL
LIN {X 0,Y 445.945,Z 211.644,A -85,B 0,C 180,E1 -8539.436,E2 -8539.436} C_VEL
LIN {X 0,Y 445.942,Z 212.333,A -85,B 0,C 180,E1 -8539.872,E2 -8539.872} C_VEL
LIN {X 0,Y 448.286,Z 222.862,A -85,B 0,C 180,E1 -8540.354,E2 -8540.354} C_VEL
LIN {X 0,Y 448.43,Z 230.258,A -85,B 0,C 180,E1 -8540.778,E2 -8540.778} C_VEL
LIN {X 0,Y 448.274,Z 237.915,A -85,B 0,C 180,E1 -8541.355,E2 -8541.355} C_VEL
LIN {X 0,Y 448.01,Z 244.556,A -85,B 0,C 180,E1 -8541.996,E2 -8541.996} C_VEL
LIN {X 0,Y 447.698,Z 250.98,A -85,B 0,C 180,E1 -8542.784,E2 -8542.784} C_VEL
LIN {X 0,Y 447.543,Z 255.455,A -85,B 0,C 180,E1 -8543.462,E2 -8543.462} C_VEL
LIN {X 0,Y 447.099,Z 261.202,A -85,B 0,C 180,E1 -8544.587,E2 -8544.587} C_VEL
LIN {X 0,Y 446.982,Z 266.047,A -85,B 0,C 180,E1 -8545.942,E2 -8545.942} C_VEL
LIN {X 0,Y 446.529,Z 269.259,A -85,B 0,C 180,E1 -8547.292,E2 -8547.292} C_VEL
LIN {X 0,Y 446.509,Z 270.584,A -85,B 0,C 180,E1 -8548.195,E2 -8548.195} C_VEL
LIN {X 0,Y 446.41,Z 271.372,A -85,B 0,C 180,E1 -8549.097,E2 -8549.097} C_VEL
LIN {X 0,Y 446.371,Z 271.644,A -85,B 0,C 180,E1 -8549.999,E2 -8549.999} C_VEL
LIN {X 0,Y 446.403,Z 271.421,A -85,B 0,C 180,E1 -8550.901,E2 -8550.901} C_VEL
LIN {X 0,Y 446.476,Z 270.691,A -85,B 0,C 180,E1 -8551.803,E2 -8551.803} C_VEL
LIN {X 0,Y 446.523,Z 269.421,A -85,B 0,C 180,E1 -8552.705,E2 -8552.705} C_VEL
LIN {X 0,Y 446.964,Z 266.314,A -85,B 0,C 180,E1 -8554.056,E2 -8554.056} C_VEL
LIN {X 0,Y 447.079,Z 261.611,A -85,B 0,C 180,E1 -8555.411,E2 -8555.411} C_VEL
LIN {X 0,Y 447.412,Z 258.435,A -85,B 0,C 180,E1 -8556.085,E2 -8556.085} C_VEL
LIN {X 0,Y 447.673,Z 251.683,A -85,B 0,C 180,E1 -8557.214,E2 -8557.214} C_VEL
LIN {X 0,Y 447.997,Z 245.419,A -85,B 0,C 180,E1 -8558.002,E2 -8558.002} C_VEL
LIN {X 0,Y 448.22,Z 239.492,A -85,B 0,C 180,E1 -8558.598,E2 -8558.598} C_VEL
LIN {X 0,Y 448.409,Z 231.987,A -85,B 0,C 180,E1 -8559.2,E2 -8559.2} C_VEL
LIN {X 0,Y 448.459,Z 224.03,A -85,B 0,C 180,E1 -8559.675,E2 -8559.675} C_VEL
LIN {X 0,Y 446.461,Z 214.581,A -85,B 0,C 180,E1 -8560.131,E2 -8560.131} C_VEL
LIN {X 0,Y 445.951,Z 212.306,A -85,B 0,C 180,E1 -8560.24,E2 -8560.24} C_VEL
LIN {X 0,Y 445.953,Z 208.487,A -85,B 0,C 180,E1 -8562.745,E2 -8562.745} C_VEL
LIN {X 0,Y 445.991,Z 203.908,A -85,B 0,C 180,E1 -8566.002,E2 -8566.002} C_VEL
LIN {X 0,Y 445.994,Z 199.588,A -85,B 0,C 180,E1 -8569.323,E2 -8569.323} C_VEL
LIN {X 0,Y 446.057,Z 195.91,A -85,B 0,C 180,E1 -8572.217,E2 -8572.217} C_VEL
LIN {X 0,Y 446.184,Z 192.297,A -85,B 0,C 180,E1 -8575.167,E2 -8575.167} C_VEL
LIN {X 0,Y 446.234,Z 188.572,A -85,B 0,C 180,E1 -8578.194,E2 -8578.194} C_VEL
LIN {X 0,Y 446.25,Z 187.902,A -85,B 0,C 180,E1 -8579.222,E2 -8579.222} C_VEL
LIN {X 0,Y 446.418,Z 187.876,A -85,B 0,C 180,E1 -8582.36,E2 -8582.36} C_VEL
LIN {X 0,Y 446.416,Z 187.88,A -85,B 0,C 180,E1 -8585.625,E2 -8585.625} C_VEL
LIN {X 0,Y 446.452,Z 187.875,A -85,B 0,C 180,E1 -8589.024,E2 -8589.024} C_VEL
LIN {X 0,Y 446.43,Z 187.873,A -85,B 0,C 180,E1 -8592.276,E2 -8592.276} C_VEL
LIN {X 0,Y 446.448,Z 187.877,A -85,B 0,C 180,E1 -8595.102,E2 -8595.102} C_VEL
LIN {X 0,Y 446.421,Z 187.879,A -85,B 0,C 180,E1 -8598.608,E2 -8598.608} C_VEL
LIN {X 0,Y 446.457,Z 187.874,A -85,B 0,C 180,E1 -8600.974,E2 -8600.974} C_VEL
LIN {X 0,Y 446.413,Z 187.879,A -85,B 0,C 180,E1 -8604.373,E2 -8604.373} C_VEL
LIN {X 0,Y 446.42,Z 187.873,A -85,B 0,C 180,E1 -8607.638,E2 -8607.638} C_VEL
LIN {X 0,Y 446.46,Z 187.869,A -85,B 0,C 180,E1 -8610.791,E2 -8610.791} C_VEL
LIN {X 0,Y 446.467,Z 187.871,A -85,B 0,C 180,E1 -8613.848,E2 -8613.848} C_VEL
LIN {X 0,Y 446.419,Z 187.874,A -85,B 0,C 180,E1 -8616.823,E2 -8616.823} C_VEL
LIN {X 0,Y 446.434,Z 187.872,A -85,B 0,C 180,E1 -8619.737,E2 -8619.737} C_VEL
LIN {X 0,Y 446.455,Z 187.87,A -85,B 0,C 180,E1 -8622.597,E2 -8622.597} C_VEL
LIN {X 0,Y 446.462,Z 187.866,A -85,B 0,C 180,E1 -8625.412,E2 -8625.412} C_VEL
LIN {X 0,Y 446.508,Z 187.862,A -85,B 0,C 180,E1 -8628.193,E2 -8628.193} C_VEL
LIN {X 0,Y 446.589,Z 187.854,A -85,B 0,C 180,E1 -8631.858,E2 -8631.858} C_VEL
LIN {X 0,Y 446.63,Z 187.845,A -85,B 0,C 180,E1 -8634.582,E2 -8634.582} C_VEL
LIN {X 0,Y 446.696,Z 187.843,A -85,B 0,C 180,E1 -8637.295,E2 -8637.295} C_VEL
LIN {X 0,Y 446.78,Z 187.822,A -85,B 0,C 180,E1 -8640,E2 -8640} C_VEL
LIN {X 0,Y 446.677,Z 187.847,A -85,B 0,C 180,E1 -8642.705,E2 -8642.705} C_VEL
LIN {X 0,Y 446.625,Z 187.849,A -85,B 0,C 180,E1 -8646.324,E2 -8646.324} C_VEL
LIN {X 0,Y 446.524,Z 187.859,A -85,B 0,C 180,E1 -8649.056,E2 -8649.056} C_VEL
LIN {X 0,Y 446.509,Z 187.862,A -85,B 0,C 180,E1 -8652.73,E2 -8652.73} C_VEL
LIN {X 0,Y 446.483,Z 187.871,A -85,B 0,C 180,E1 -8656.228,E2 -8656.228} C_VEL
LIN {X 0,Y 446.456,Z 187.871,A -85,B 0,C 180,E1 -8659.304,E2 -8659.304} C_VEL
LIN {X 0,Y 446.404,Z 187.881,A -85,B 0,C 180,E1 -8662.2,E2 -8662.2} C_VEL
LIN {X 0,Y 446.409,Z 187.878,A -85,B 0,C 180,E1 -8665.155,E2 -8665.155} C_VEL
LIN {X 0,Y 446.405,Z 187.879,A -85,B 0,C 180,E1 -8668.184,E2 -8668.184} C_VEL
LIN {X 0,Y 446.404,Z 187.881,A -85,B 0,C 180,E1 -8671.301,E2 -8671.301} C_VEL
LIN {X 0,Y 446.412,Z 187.873,A -85,B 0,C 180,E1 -8674.525,E2 -8674.525} C_VEL
LIN {X 0,Y 446.4,Z 187.88,A -85,B 0,C 180,E1 -8678.079,E2 -8678.079} C_VEL
LIN {X 0,Y 446.401,Z 187.875,A -85,B 0,C 180,E1 -8681.394,E2 -8681.394} C_VEL
LIN {X 0,Y 446.443,Z 187.875,A -85,B 0,C 180,E1 -8685.105,E2 -8685.105} C_VEL
LIN {X 0,Y 446.421,Z 187.873,A -85,B 0,C 180,E1 -8688.61,E2 -8688.61} C_VEL
LIN {X 0,Y 446.438,Z 187.871,A -85,B 0,C 180,E1 -8690.974,E2 -8690.974} C_VEL
LIN {X 0,Y 446.423,Z 187.921,A -85,B 0,C 180,E1 -8693.959,E2 -8693.959} C_VEL
LIN {X 0,Y 449.041,Z 198.955,A -85,B 0,C 180,E1 -8696.786,E2 -8696.786} C_VEL
LIN {X 0,Y 451.189,Z 208.584,A -85,B 0,C 180,E1 -8699.069,E2 -8699.069} C_VEL
LIN {X 0,Y 451.377,Z 212.253,A -85,B 0,C 180,E1 -8699.86,E2 -8699.86} C_VEL
LIN {X 0,Y 449.811,Z 229.632,A -85,B 0,C 180,E1 -8703.309,E2 -8703.309} C_VEL
LIN {X 0,Y 448.538,Z 247.197,A -85,B 0,C 180,E1 -8706.696,E2 -8706.696} C_VEL
LIN {X 0,Y 447.573,Z 263.429,A -85,B 0,C 180,E1 -8709.792,E2 -8709.792} C_VEL
LIN {X 0,Y 446.642,Z 281.543,A -85,B 0,C 180,E1 -8713.313,E2 -8713.313} C_VEL
LIN {X 0,Y 446.491,Z 285.781,A -85,B 0,C 180,E1 -8714.128,E2 -8714.128} C_VEL
LIN {X 0,Y 448.057,Z 301.864,A -85,B 0,C 180,E1 -8714.551,E2 -8714.551} C_VEL
LIN {X 0,Y 448.601,Z 312.906,A -85,B 0,C 180,E1 -8714.962,E2 -8714.962} C_VEL
LIN {X 0,Y 448.211,Z 325.698,A -85,B 0,C 180,E1 -8715.588,E2 -8715.588} C_VEL
LIN {X 0,Y 447.661,Z 337.842,A -85,B 0,C 180,E1 -8716.381,E2 -8716.381} C_VEL
LIN {X 0,Y 447.145,Z 348.809,A -85,B 0,C 180,E1 -8717.29,E2 -8717.29} C_VEL
LIN {X 0,Y 446.753,Z 357.748,A -85,B 0,C 180,E1 -8718.201,E2 -8718.201} C_VEL
LIN {X 0,Y 446.303,Z 366.941,A -85,B 0,C 180,E1 -8719.338,E2 -8719.338} C_VEL
LIN {X 0,Y 445.955,Z 375.895,A -85,B 0,C 180,E1 -8720.705,E2 -8720.705} C_VEL
LIN {X 0,Y 445.721,Z 383.058,A -85,B 0,C 180,E1 -8722.071,E2 -8722.071} C_VEL
LIN {X 0,Y 445.568,Z 389.218,A -85,B 0,C 180,E1 -8723.57,E2 -8723.57} C_VEL
LIN {X 0,Y 445.589,Z 393.792,A -85,B 0,C 180,E1 -8725.025,E2 -8725.025} C_VEL
LIN {X 0,Y 445.589,Z 396.913,A -85,B 0,C 180,E1 -8726.384,E2 -8726.384} C_VEL
LIN {X 0,Y 445.577,Z 398.438,A -85,B 0,C 180,E1 -8727.289,E2 -8727.289} C_VEL
LIN {X 0,Y 445.595,Z 399.483,A -85,B 0,C 180,E1 -8728.194,E2 -8728.194} C_VEL
LIN {X 0,Y 445.552,Z 400.111,A -85,B 0,C 180,E1 -8729.097,E2 -8729.097} C_VEL
LIN {X 0,Y 445.552,Z 400.333,A -85,B 0,C 180,E1 -8730.001,E2 -8730.001} C_VEL
LIN {X 0,Y 445.554,Z 400.109,A -85,B 0,C 180,E1 -8730.905,E2 -8730.905} C_VEL
LIN {X 0,Y 445.584,Z 399.447,A -85,B 0,C 180,E1 -8731.809,E2 -8731.809} C_VEL
LIN {X 0,Y 445.583,Z 398.372,A -85,B 0,C 180,E1 -8732.713,E2 -8732.713} C_VEL
LIN {X 0,Y 445.603,Z 396.871,A -85,B 0,C 180,E1 -8733.618,E2 -8733.618} C_VEL
LIN {X 0,Y 445.596,Z 393.735,A -85,B 0,C 180,E1 -8734.978,E2 -8734.978} C_VEL
LIN {X 0,Y 445.587,Z 389.087,A -85,B 0,C 180,E1 -8736.451,E2 -8736.451} C_VEL
LIN {X 0,Y 445.737,Z 382.992,A -85,B 0,C 180,E1 -8737.931,E2 -8737.931} C_VEL
LIN {X 0,Y 445.998,Z 375.921,A -85,B 0,C 180,E1 -8739.296,E2 -8739.296} C_VEL
LIN {X 0,Y 446.33,Z 367.109,A -85,B 0,C 180,E1 -8740.663,E2 -8740.663} C_VEL
LIN {X 0,Y 446.781,Z 358.122,A -85,B 0,C 180,E1 -8741.801,E2 -8741.801} C_VEL
LIN {X 0,Y 447.214,Z 347.281,A -85,B 0,C 180,E1 -8742.927,E2 -8742.927} C_VEL
LIN {X 0,Y 447.984,Z 334.621,A -85,B 0,C 180,E1 -8743.959,E2 -8743.959} C_VEL
LIN {X 0,Y 448.615,Z 322.187,A -85,B 0,C 180,E1 -8744.749,E2 -8744.749} C_VEL
LIN {X 0,Y 448.943,Z 310.591,A -85,B 0,C 180,E1 -8745.319,E2 -8745.319} C_VEL
LIN {X 0,Y 448.138,Z 296.611,A -85,B 0,C 180,E1 -8745.862,E2 -8745.862} C_VEL
LIN {X 0,Y 446.574,Z 283.585,A -85,B 0,C 180,E1 -8746.278,E2 -8746.278} C_VEL
LIN {X 0,Y 447.412,Z 265.518,A -85,B 0,C 180,E1 -8749.801,E2 -8749.801} C_VEL
LIN {X 0,Y 448.363,Z 249.582,A -85,B 0,C 180,E1 -8752.847,E2 -8752.847} C_VEL
LIN {X 0,Y 449.485,Z 233.323,A -85,B 0,C 180,E1 -8755.965,E2 -8755.965} C_VEL
LIN {X 0,Y 450.896,Z 216.821,A -85,B 0,C 180,E1 -8759.207,E2 -8759.207} C_VEL
LIN {X 0,Y 451.392,Z 210.959,A -85,B 0,C 180,E1 -8760.4,E2 -8760.4} C_VEL
LIN {X 0,Y 450.636,Z 206.088,A -85,B 0,C 180,E1 -8761.498,E2 -8761.498} C_VEL
LIN {X 0,Y 447.574,Z 192.608,A -85,B 0,C 180,E1 -8764.79,E2 -8764.79} C_VEL
LIN {X 0,Y 446.438,Z 187.879,A -85,B 0,C 180,E1 -8766.077,E2 -8766.077} C_VEL
LIN {X 0,Y 446.44,Z 187.876,A -85,B 0,C 180,E1 -8769.522,E2 -8769.522} C_VEL
LIN {X 0,Y 446.434,Z 187.875,A -85,B 0,C 180,E1 -8772.605,E2 -8772.605} C_VEL
LIN {X 0,Y 446.457,Z 187.873,A -85,B 0,C 180,E1 -8775.104,E2 -8775.104} C_VEL
LIN {X 0,Y 446.433,Z 187.877,A -85,B 0,C 180,E1 -8778.609,E2 -8778.609} C_VEL
LIN {X 0,Y 446.429,Z 187.88,A -85,B 0,C 180,E1 -8780.971,E2 -8780.971} C_VEL
LIN {X 0,Y 446.437,Z 187.919,A -85,B 0,C 180,E1 -8782.267,E2 -8782.267} C_VEL
LIN {X 0,Y 447.82,Z 194.478,A -85,B 0,C 180,E1 -8784.695,E2 -8784.695} C_VEL
LIN {X 0,Y 448.006,Z 198.9,A -85,B 0,C 180,E1 -8786.247,E2 -8786.247} C_VEL
LIN {X 0,Y 447.567,Z 209.298,A -85,B 0,C 180,E1 -8789.835,E2 -8789.835} C_VEL
LIN {X 0,Y 447.446,Z 215.004,A -85,B 0,C 180,E1 -8791.887,E2 -8791.887} C_VEL
LIN {X 0,Y 447.251,Z 223.332,A -85,B 0,C 180,E1 -8794.895,E2 -8794.895} C_VEL
LIN {X 0,Y 447.05,Z 231.995,A -85,B 0,C 180,E1 -8798.055,E2 -8798.055} C_VEL
LIN {X 0,Y 446.857,Z 240.447,A -85,B 0,C 180,E1 -8801.191,E2 -8801.191} C_VEL
LIN {X 0,Y 446.683,Z 247.279,A -85,B 0,C 180,E1 -8803.733,E2 -8803.733} C_VEL
LIN {X 0,Y 449.668,Z 259.476,A -85,B 0,C 180,E1 -8804.275,E2 -8804.275} C_VEL
LIN {X 0,Y 450.165,Z 263.715,A -85,B 0,C 180,E1 -8804.474,E2 -8804.474} C_VEL
LIN {X 0,Y 449.58,Z 277.454,A -85,B 0,C 180,E1 -8805.168,E2 -8805.168} C_VEL
LIN {X 0,Y 449.057,Z 289.074,A -85,B 0,C 180,E1 -8805.943,E2 -8805.943} C_VEL
LIN {X 0,Y 448.401,Z 301.208,A -85,B 0,C 180,E1 -8806.979,E2 -8806.979} C_VEL
LIN {X 0,Y 447.805,Z 310.85,A -85,B 0,C 180,E1 -8807.998,E2 -8807.998} C_VEL
LIN {X 0,Y 447.245,Z 319.621,A -85,B 0,C 180,E1 -8809.131,E2 -8809.131} C_VEL
LIN {X 0,Y 446.82,Z 328.192,A -85,B 0,C 180,E1 -8810.494,E2 -8810.494} C_VEL
LIN {X 0,Y 446.343,Z 335.12,A -85,B 0,C 180,E1 -8811.853,E2 -8811.853} C_VEL
LIN {X 0,Y 446.051,Z 341.097,A -85,B 0,C 180,E1 -8813.354,E2 -8813.354} C_VEL
LIN {X 0,Y 445.768,Z 346.12,A -85,B 0,C 180,E1 -8815.025,E2 -8815.025} C_VEL
LIN {X 0,Y 445.675,Z 348.998,A -85,B 0,C 180,E1 -8816.384,E2 -8816.384} C_VEL
LIN {X 0,Y 445.623,Z 350.367,A -85,B 0,C 180,E1 -8817.288,E2 -8817.288} C_VEL
LIN {X 0,Y 445.526,Z 351.316,A -85,B 0,C 180,E1 -8818.192,E2 -8818.192} C_VEL
LIN {X 0,Y 445.437,Z 351.874,A -85,B 0,C 180,E1 -8819.096,E2 -8819.096} C_VEL
LIN {X 0,Y 445.412,Z 352.026,A -85,B 0,C 180,E1 -8820,E2 -8820} C_VEL
LIN {X 0,Y 445.435,Z 351.732,A -85,B 0,C 180,E1 -8820.904,E2 -8820.904} C_VEL
LIN {X 0,Y 445.56,Z 349.965,A -85,B 0,C 180,E1 -8822.712,E2 -8822.712} C_VEL
LIN {X 0,Y 445.651,Z 348.435,A -85,B 0,C 180,E1 -8823.617,E2 -8823.617} C_VEL
LIN {X 0,Y 445.618,Z 345.334,A -85,B 0,C 180,E1 -8824.976,E2 -8824.976} C_VEL
LIN {X 0,Y 445.874,Z 341.15,A -85,B 0,C 180,E1 -8826.335,E2 -8826.335} C_VEL
LIN {X 0,Y 446.076,Z 334.773,A -85,B 0,C 180,E1 -8827.924,E2 -8827.924} C_VEL
LIN {X 0,Y 446.481,Z 327.811,A -85,B 0,C 180,E1 -8829.285,E2 -8829.285} C_VEL
LIN {X 0,Y 446.913,Z 319.104,A -85,B 0,C 180,E1 -8830.648,E2 -8830.648} C_VEL
LIN {X 0,Y 447.462,Z 309.254,A -85,B 0,C 180,E1 -8831.897,E2 -8831.897} C_VEL
LIN {X 0,Y 447.974,Z 298.751,A -85,B 0,C 180,E1 -8832.967,E2 -8832.967} C_VEL
LIN {X 0,Y 448.459,Z 286.88,A -85,B 0,C 180,E1 -8833.943,E2 -8833.943} C_VEL
LIN {X 0,Y 449.006,Z 274.305,A -85,B 0,C 180,E1 -8834.735,E2 -8834.735} C_VEL
LIN {X 0,Y 449.395,Z 261.181,A -85,B 0,C 180,E1 -8835.36,E2 -8835.36} C_VEL
LIN {X 0,Y 446.699,Z 247.322,A -85,B 0,C 180,E1 -8835.901,E2 -8835.901} C_VEL
LIN {X 0,Y 446.259,Z 244.849,A -85,B 0,C 180,E1 -8836.007,E2 -8836.007} C_VEL
LIN {X 0,Y 446.41,Z 236.043,A -85,B 0,C 180,E1 -8839.306,E2 -8839.306} C_VEL
LIN {X 0,Y 446.587,Z 227.094,A -85,B 0,C 180,E1 -8842.679,E2 -8842.679} C_VEL
LIN {X 0,Y 446.734,Z 219.265,A -85,B 0,C 180,E1 -8845.635,E2 -8845.635} C_VEL
LIN {X 0,Y 446.946,Z 211.219,A -85,B 0,C 180,E1 -8848.674,E2 -8848.674} C_VEL
LIN {X 0,Y 447.117,Z 204.429,A -85,B 0,C 180,E1 -8851.246,E2 -8851.246} C_VEL
LIN {X 0,Y 447.243,Z 195.99,A -85,B 0,C 180,E1 -8854.452,E2 -8854.452} C_VEL
LIN {X 0,Y 447.073,Z 191.643,A -85,B 0,C 180,E1 -8856.106,E2 -8856.106} C_VEL
LIN {X 0,Y 446.482,Z 187.872,A -85,B 0,C 180,E1 -8857.587,E2 -8857.587} C_VEL
LIN {X 0,Y 446.428,Z 187.879,A -85,B 0,C 180,E1 -8860.917,E2 -8860.917} C_VEL
LIN {X 0,Y 446.403,Z 187.879,A -85,B 0,C 180,E1 -8863.846,E2 -8863.846} C_VEL
LIN {X 0,Y 446.402,Z 187.879,A -85,B 0,C 180,E1 -8866.403,E2 -8866.403} C_VEL
LIN {X 0,Y 446.432,Z 187.878,A -85,B 0,C 180,E1 -8869.082,E2 -8869.082} C_VEL
LIN {X 0,Y 446.398,Z 187.884,A -85,B 0,C 180,E1 -8872.119,E2 -8872.119} C_VEL
LIN {X 0,Y 446.425,Z 187.881,A -85,B 0,C 180,E1 -8875.476,E2 -8875.476} C_VEL
LIN {X 0,Y 446.393,Z 187.884,A -85,B 0,C 180,E1 -8878.697,E2 -8878.697} C_VEL
LIN {X 0,Y 446.268,Z 187.9,A -85,B 0,C 180,E1 -8880.777,E2 -8880.777} C_VEL
LIN {X 0,Y 446.245,Z 188.526,A -85,B 0,C 180,E1 -8881.88,E2 -8881.88} C_VEL
LIN {X 0,Y 446.192,Z 192.151,A -85,B 0,C 180,E1 -8884.831,E2 -8884.831} C_VEL
LIN {X 0,Y 446.083,Z 196.503,A -85,B 0,C 180,E1 -8888.364,E2 -8888.364} C_VEL
LIN {X 0,Y 446.004,Z 200.665,A -85,B 0,C 180,E1 -8891.629,E2 -8891.629} C_VEL
LIN {X 0,Y 445.982,Z 204.397,A -85,B 0,C 180,E1 -8894.46,E2 -8894.46} C_VEL
LIN {X 0,Y 446.03,Z 209.704,A -85,B 0,C 180,E1 -8898.179,E2 -8898.179} C_VEL
LIN {X 0,Y 445.945,Z 211.644,A -85,B 0,C 180,E1 -8899.436,E2 -8899.436} C_VEL
LIN {X 0,Y 445.924,Z 212.92,A -85,B 0,C 180,E1 -8899.72,E2 -8899.72} C_VEL
LIN {X 0,Y 445.82,Z 215.785,A -85,B 0,C 180,E1 -8899.962,E2 -8899.962} C_VEL
LIN {X 0,Y 445.075,Z 223.983,A -85,B 0,C 180,E1 -8900.302,E2 -8900.302} C_VEL
LIN {X 0,Y 442.116,Z 235.315,A -85,B 0,C 180,E1 -8900.896,E2 -8900.896} C_VEL
LIN {X 0,Y 441.338,Z 239.701,A -85,B 0,C 180,E1 -8901.27,E2 -8901.27} C_VEL
LIN {X 0,Y 441.029,Z 246.728,A -85,B 0,C 180,E1 -8901.984,E2 -8901.984} C_VEL
LIN {X 0,Y 440.784,Z 253.688,A -85,B 0,C 180,E1 -8902.901,E2 -8902.901} C_VEL
LIN {X 0,Y 440.47,Z 258.988,A -85,B 0,C 180,E1 -8903.816,E2 -8903.816} C_VEL
LIN {X 0,Y 440.107,Z 262.23,A -85,B 0,C 180,E1 -8904.501,E2 -8904.501} C_VEL
LIN {X 0,Y 439.987,Z 267.044,A -85,B 0,C 180,E1 -8905.877,E2 -8905.877} C_VEL
LIN {X 0,Y 439.516,Z 270.242,A -85,B 0,C 180,E1 -8907.249,E2 -8907.249} C_VEL
LIN {X 0,Y 439.492,Z 271.562,A -85,B 0,C 180,E1 -8908.166,E2 -8908.166} C_VEL
LIN {X 0,Y 439.389,Z 272.347,A -85,B 0,C 180,E1 -8909.082,E2 -8909.082} C_VEL
LIN {X 0,Y 439.348,Z 272.618,A -85,B 0,C 180,E1 -8909.999,E2 -8909.999} C_VEL
LIN {X 0,Y 439.382,Z 272.395,A -85,B 0,C 180,E1 -8910.915,E2 -8910.915} C_VEL
LIN {X 0,Y 439.462,Z 271.666,A -85,B 0,C 180,E1 -8911.832,E2 -8911.832} C_VEL
LIN {X 0,Y 439.509,Z 270.402,A -85,B 0,C 180,E1 -8912.748,E2 -8912.748} C_VEL
LIN {X 0,Y 439.971,Z 267.307,A -85,B 0,C 180,E1 -8914.121,E2 -8914.121} C_VEL
LIN {X 0,Y 440.084,Z 262.628,A -85,B 0,C 180,E1 -8915.497,E2 -8915.497} C_VEL
LIN {X 0,Y 440.433,Z 259.474,A -85,B 0,C 180,E1 -8916.182,E2 -8916.182} C_VEL
LIN {X 0,Y 440.715,Z 252.78,A -85,B 0,C 180,E1 -8917.328,E2 -8917.328} C_VEL
LIN {X 0,Y 441.067,Z 246.563,A -85,B 0,C 180,E1 -8918.128,E2 -8918.128} C_VEL
LIN {X 0,Y 441.305,Z 240.278,A -85,B 0,C 180,E1 -8918.773,E2 -8918.773} C_VEL
LIN {X 0,Y 441.5,Z 233.034,A -85,B 0,C 180,E1 -8919.366,E2 -8919.366} C_VEL
LIN {X 0,Y 441.551,Z 225.112,A -85,B 0,C 180,E1 -8919.85,E2 -8919.85} C_VEL
LIN {X 0,Y 439.498,Z 215.531,A -85,B 0,C 180,E1 -8920.328,E2 -8920.328} C_VEL
LIN {X 0,Y 438.921,Z 212.942,A -85,B 0,C 180,E1 -8920.435,E2 -8920.435} C_VEL
LIN {X 0,Y 438.921,Z 209.112,A -85,B 0,C 180,E1 -8922.953,E2 -8922.953} C_VEL
LIN {X 0,Y 438.954,Z 204.664,A -85,B 0,C 180,E1 -8926.126,E2 -8926.126} C_VEL
LIN {X 0,Y 438.937,Z 200.1,A -85,B 0,C 180,E1 -8929.646,E2 -8929.646} C_VEL
LIN {X 0,Y 439.028,Z 196.358,A -85,B 0,C 180,E1 -8932.592,E2 -8932.592} C_VEL
LIN {X 0,Y 439.139,Z 192.7,A -85,B 0,C 180,E1 -8935.6,E2 -8935.6} C_VEL
LIN {X 0,Y 439.155,Z 188.907,A -85,B 0,C 180,E1 -8938.691,E2 -8938.691} C_VEL
LIN {X 0,Y 439.319,Z 188.76,A -85,B 0,C 180,E1 -8940.79,E2 -8940.79} C_VEL
LIN {X 0,Y 439.383,Z 188.754,A -85,B 0,C 180,E1 -8944.042,E2 -8944.042} C_VEL
LIN {X 0,Y 439.352,Z 188.757,A -85,B 0,C 180,E1 -8946.887,E2 -8946.887} C_VEL
LIN {X 0,Y 439.401,Z 188.75,A -85,B 0,C 180,E1 -8949.849,E2 -8949.849} C_VEL
LIN {X 0,Y 439.38,Z 188.753,A -85,B 0,C 180,E1 -8952.626,E2 -8952.626} C_VEL
LIN {X 0,Y 439.395,Z 188.753,A -85,B 0,C 180,E1 -8955.27,E2 -8955.27} C_VEL
LIN {X 0,Y 439.381,Z 188.755,A -85,B 0,C 180,E1 -8958.742,E2 -8958.742} C_VEL
LIN {X 0,Y 439.379,Z 188.751,A -85,B 0,C 180,E1 -8961.604,E2 -8961.604} C_VEL
LIN {X 0,Y 439.393,Z 188.752,A -85,B 0,C 180,E1 -8964.843,E2 -8964.843} C_VEL
LIN {X 0,Y 439.379,Z 188.754,A -85,B 0,C 180,E1 -8968.14,E2 -8968.14} C_VEL
LIN {X 0,Y 439.416,Z 188.744,A -85,B 0,C 180,E1 -8971.326,E2 -8971.326} C_VEL
LIN {X 0,Y 439.395,Z 188.747,A -85,B 0,C 180,E1 -8974.414,E2 -8974.414} C_VEL
LIN {X 0,Y 439.355,Z 188.755,A -85,B 0,C 180,E1 -8977.424,E2 -8977.424} C_VEL
LIN {X 0,Y 439.431,Z 188.743,A -85,B 0,C 180,E1 -8980.662,E2 -8980.662} C_VEL
LIN {X 0,Y 439.464,Z 188.736,A -85,B 0,C 180,E1 -8984.224,E2 -8984.224} C_VEL
LIN {X 0,Y 439.473,Z 188.74,A -85,B 0,C 180,E1 -8988.001,E2 -8988.001} C_VEL
LIN {X 0,Y 439.537,Z 188.734,A -85,B 0,C 180,E1 -8991.726,E2 -8991.726} C_VEL
LIN {X 0,Y 439.605,Z 188.72,A -85,B 0,C 180,E1 -8994.496,E2 -8994.496} C_VEL
LIN {X 0,Y 439.625,Z 188.72,A -85,B 0,C 180,E1 -8998.168,E2 -8998.168} C_VEL
LIN {X 0,Y 439.75,Z 188.698,A -85,B 0,C 180,E1 -9000,E2 -9000} C_VEL
LIN {X 0,Y 439.626,Z 188.726,A -85,B 0,C 180,E1 -9002.749,E2 -9002.749} C_VEL
LIN {X 0,Y 439.6,Z 188.725,A -85,B 0,C 180,E1 -9006.425,E2 -9006.425} C_VEL
LIN {X 0,Y 439.486,Z 188.734,A -85,B 0,C 180,E1 -9009.202,E2 -9009.202} C_VEL
LIN {X 0,Y 439.453,Z 188.739,A -85,B 0,C 180,E1 -9012.938,E2 -9012.938} C_VEL
LIN {X 0,Y 439.434,Z 188.747,A -85,B 0,C 180,E1 -9016.348,E2 -9016.348} C_VEL
LIN {X 0,Y 439.39,Z 188.753,A -85,B 0,C 180,E1 -9019.627,E2 -9019.627} C_VEL
LIN {X 0,Y 439.35,Z 188.757,A -85,B 0,C 180,E1 -9022.576,E2 -9022.576} C_VEL
LIN {X 0,Y 439.355,Z 188.76,A -85,B 0,C 180,E1 -9025.588,E2 -9025.588} C_VEL
LIN {X 0,Y 439.37,Z 188.754,A -85,B 0,C 180,E1 -9028.677,E2 -9028.677} C_VEL
LIN {X 0,Y 439.358,Z 188.756,A -85,B 0,C 180,E1 -9032.031,E2 -9032.031} C_VEL
LIN {X 0,Y 439.381,Z 188.755,A -85,B 0,C 180,E1 -9035.341,E2 -9035.341} C_VEL
LIN {X 0,Y 439.358,Z 188.758,A -85,B 0,C 180,E1 -9038.598,E2 -9038.598} C_VEL
LIN {X 0,Y 439.361,Z 188.75,A -85,B 0,C 180,E1 -9041.255,E2 -9041.255} C_VEL
LIN {X 0,Y 439.391,Z 188.755,A -85,B 0,C 180,E1 -9044.731,E2 -9044.731} C_VEL
LIN {X 0,Y 439.389,Z 188.744,A -85,B 0,C 180,E1 -9047.797,E2 -9047.797} C_VEL
LIN {X 0,Y 439.42,Z 188.747,A -85,B 0,C 180,E1 -9050.229,E2 -9050.229} C_VEL
LIN {X 0,Y 439.405,Z 188.933,A -85,B 0,C 180,E1 -9053.569,E2 -9053.569} C_VEL
LIN {X 0,Y 442.021,Z 199.952,A -85,B 0,C 180,E1 -9056.462,E2 -9056.462} C_VEL
LIN {X 0,Y 444.408,Z 210.866,A -85,B 0,C 180,E1 -9059.1,E2 -9059.1} C_VEL
LIN {X 0,Y 444.441,Z 214.418,A -85,B 0,C 180,E1 -9059.865,E2 -9059.865} C_VEL
LIN {X 0,Y 442.907,Z 230.468,A -85,B 0,C 180,E1 -9063.114,E2 -9063.114} C_VEL
LIN {X 0,Y 441.564,Z 247.883,A -85,B 0,C 180,E1 -9066.554,E2 -9066.554} C_VEL
LIN {X 0,Y 440.453,Z 265.455,A -85,B 0,C 180,E1 -9069.987,E2 -9069.987} C_VEL
LIN {X 0,Y 439.58,Z 281.93,A -85,B 0,C 180,E1 -9073.276,E2 -9073.276} C_VEL
LIN {X 0,Y 439.445,Z 284.901,A -85,B 0,C 180,E1 -9073.878,E2 -9073.878} C_VEL
LIN {X 0,Y 441.139,Z 302.759,A -85,B 0,C 180,E1 -9074.376,E2 -9074.376} C_VEL
LIN {X 0,Y 441.62,Z 314.416,A -85,B 0,C 180,E1 -9074.837,E2 -9074.837} C_VEL
LIN {X 0,Y 441.191,Z 326.598,A -85,B 0,C 180,E1 -9075.471,E2 -9075.471} C_VEL
LIN {X 0,Y 440.645,Z 338.586,A -85,B 0,C 180,E1 -9076.286,E2 -9076.286} C_VEL
LIN {X 0,Y 440.118,Z 349.22,A -85,B 0,C 180,E1 -9077.201,E2 -9077.201} C_VEL
LIN {X 0,Y 439.622,Z 358.985,A -85,B 0,C 180,E1 -9078.24,E2 -9078.24} C_VEL
LIN {X 0,Y 439.188,Z 367.906,A -85,B 0,C 180,E1 -9079.397,E2 -9079.397} C_VEL
LIN {X 0,Y 438.85,Z 376.607,A -85,B 0,C 180,E1 -9080.786,E2 -9080.786} C_VEL
LIN {X 0,Y 438.611,Z 383.522,A -85,B 0,C 180,E1 -9082.173,E2 -9082.173} C_VEL
LIN {X 0,Y 438.474,Z 389.159,A -85,B 0,C 180,E1 -9083.596,E2 -9083.596} C_VEL
LIN {X 0,Y 438.513,Z 393.308,A -85,B 0,C 180,E1 -9084.944,E2 -9084.944} C_VEL
LIN {X 0,Y 438.489,Z 396.458,A -85,B 0,C 180,E1 -9086.325,E2 -9086.325} C_VEL
LIN {X 0,Y 438.499,Z 398.002,A -85,B 0,C 180,E1 -9087.245,E2 -9087.245} C_VEL
LIN {X 0,Y 438.502,Z 399.066,A -85,B 0,C 180,E1 -9088.164,E2 -9088.164} C_VEL
LIN {X 0,Y 438.485,Z 399.703,A -85,B 0,C 180,E1 -9089.083,E2 -9089.083} C_VEL
LIN {X 0,Y 438.481,Z 399.934,A -85,B 0,C 180,E1 -9090.001,E2 -9090.001} C_VEL
LIN {X 0,Y 438.486,Z 399.729,A -85,B 0,C 180,E1 -9090.92,E2 -9090.92} C_VEL
LIN {X 0,Y 438.493,Z 399.071,A -85,B 0,C 180,E1 -9091.838,E2 -9091.838} C_VEL
LIN {X 0,Y 438.505,Z 398.003,A -85,B 0,C 180,E1 -9092.757,E2 -9092.757} C_VEL
LIN {X 0,Y 438.499,Z 396.513,A -85,B 0,C 180,E1 -9093.677,E2 -9093.677} C_VEL
LIN {X 0,Y 438.521,Z 393.394,A -85,B 0,C 180,E1 -9095.058,E2 -9095.058} C_VEL
LIN {X 0,Y 438.507,Z 389.172,A -85,B 0,C 180,E1 -9096.443,E2 -9096.443} C_VEL
LIN {X 0,Y 438.677,Z 382.689,A -85,B 0,C 180,E1 -9098.06,E2 -9098.06} C_VEL
LIN {X 0,Y 438.934,Z 375.65,A -85,B 0,C 180,E1 -9099.447,E2 -9099.447} C_VEL
LIN {X 0,Y 439.235,Z 368.497,A -85,B 0,C 180,E1 -9100.604,E2 -9100.604} C_VEL
LIN {X 0,Y 439.688,Z 359.927,A -85,B 0,C 180,E1 -9101.76,E2 -9101.76} C_VEL
LIN {X 0,Y 440.147,Z 349.426,A -85,B 0,C 180,E1 -9102.918,E2 -9102.918} C_VEL
LIN {X 0,Y 440.909,Z 337.777,A -85,B 0,C 180,E1 -9103.952,E2 -9103.952} C_VEL
LIN {X 0,Y 441.554,Z 326.367,A -85,B 0,C 180,E1 -9104.755,E2 -9104.755} C_VEL
LIN {X 0,Y 442.241,Z 312.687,A -85,B 0,C 180,E1 -9105.498,E2 -9105.498} C_VEL
LIN {X 0,Y 441.551,Z 298.884,A -85,B 0,C 180,E1 -9106.08,E2 -9106.08} C_VEL
LIN {X 0,Y 439.541,Z 282.334,A -85,B 0,C 180,E1 -9106.637,E2 -9106.637} C_VEL
LIN {X 0,Y 440.402,Z 265.388,A -85,B 0,C 180,E1 -9110.018,E2 -9110.018} C_VEL
LIN {X 0,Y 441.376,Z 250.359,A -85,B 0,C 180,E1 -9112.962,E2 -9112.962} C_VEL
LIN {X 0,Y 442.7,Z 232.87,A -85,B 0,C 180,E1 -9116.393,E2 -9116.393} C_VEL
LIN {X 0,Y 444.323,Z 215.561,A -85,B 0,C 180,E1 -9119.885,E2 -9119.885} C_VEL
LIN {X 0,Y 444.41,Z 210.816,A -85,B 0,C 180,E1 -9120.898,E2 -9120.898} C_VEL
LIN {X 0,Y 441.693,Z 198.666,A -85,B 0,C 180,E1 -9123.843,E2 -9123.843} C_VEL
LIN {X 0,Y 439.385,Z 188.758,A -85,B 0,C 180,E1 -9126.473,E2 -9126.473} C_VEL
LIN {X 0,Y 439.407,Z 188.751,A -85,B 0,C 180,E1 -9129.85,E2 -9129.85} C_VEL
LIN {X 0,Y 439.387,Z 188.753,A -85,B 0,C 180,E1 -9132.627,E2 -9132.627} C_VEL
LIN {X 0,Y 439.405,Z 188.752,A -85,B 0,C 180,E1 -9135.271,E2 -9135.271} C_VEL
LIN {X 0,Y 439.394,Z 188.755,A -85,B 0,C 180,E1 -9138.744,E2 -9138.744} C_VEL
LIN {X 0,Y 439.407,Z 188.962,A -85,B 0,C 180,E1 -9141.691,E2 -9141.691} C_VEL
LIN {X 0,Y 440.954,Z 195.892,A -85,B 0,C 180,E1 -9144.376,E2 -9144.376} C_VEL
LIN {X 0,Y 441.231,Z 200.692,A -85,B 0,C 180,E1 -9146.118,E2 -9146.118} C_VEL
LIN {X 0,Y 440.724,Z 210.077,A -85,B 0,C 180,E1 -9149.443,E2 -9149.443} C_VEL
LIN {X 0,Y 440.605,Z 217.118,A -85,B 0,C 180,E1 -9151.93,E2 -9151.93} C_VEL
LIN {X 0,Y 440.308,Z 226.628,A -85,B 0,C 180,E1 -9155.481,E2 -9155.481} C_VEL
LIN {X 0,Y 440.073,Z 234.612,A -85,B 0,C 180,E1 -9158.45,E2 -9158.45} C_VEL
LIN {X 0,Y 439.884,Z 242.382,A -85,B 0,C 180,E1 -9161.365,E2 -9161.365} C_VEL
LIN {X 0,Y 439.773,Z 247.959,A -85,B 0,C 180,E1 -9163.399,E2 -9163.399} C_VEL
LIN {X 0,Y 442.801,Z 259.771,A -85,B 0,C 180,E1 -9163.953,E2 -9163.953} C_VEL
LIN {X 0,Y 443.438,Z 263.268,A -85,B 0,C 180,E1 -9164.134,E2 -9164.134} C_VEL
LIN {X 0,Y 443.018,Z 274.899,A -85,B 0,C 180,E1 -9164.708,E2 -9164.708} C_VEL
LIN {X 0,Y 442.413,Z 287.165,A -85,B 0,C 180,E1 -9165.501,E2 -9165.501} C_VEL
LIN {X 0,Y 441.802,Z 298.507,A -85,B 0,C 180,E1 -9166.43,E2 -9166.43} C_VEL
LIN {X 0,Y 441.043,Z 309.642,A -85,B 0,C 180,E1 -9167.577,E2 -9167.577} C_VEL
LIN {X 0,Y 440.432,Z 318.73,A -85,B 0,C 180,E1 -9168.728,E2 -9168.728} C_VEL
LIN {X 0,Y 439.962,Z 326.229,A -85,B 0,C 180,E1 -9169.88,E2 -9169.88} C_VEL
LIN {X 0,Y 439.482,Z 333.569,A -85,B 0,C 180,E1 -9171.262,E2 -9171.262} C_VEL
LIN {X 0,Y 439.123,Z 339.471,A -85,B 0,C 180,E1 -9172.644,E2 -9172.644} C_VEL
LIN {X 0,Y 438.794,Z 344.136,A -85,B 0,C 180,E1 -9174.024,E2 -9174.024} C_VEL
LIN {X 0,Y 438.751,Z 347.664,A -85,B 0,C 180,E1 -9175.406,E2 -9175.406} C_VEL
LIN {X 0,Y 438.619,Z 349.477,A -85,B 0,C 180,E1 -9176.325,E2 -9176.325} C_VEL
LIN {X 0,Y 438.546,Z 350.82,A -85,B 0,C 180,E1 -9177.244,E2 -9177.244} C_VEL
LIN {X 0,Y 438.471,Z 351.751,A -85,B 0,C 180,E1 -9178.163,E2 -9178.163} C_VEL
LIN {X 0,Y 438.376,Z 352.295,A -85,B 0,C 180,E1 -9179.081,E2 -9179.081} C_VEL
LIN {X 0,Y 438.35,Z 352.42,A -85,B 0,C 180,E1 -9180,E2 -9180} C_VEL
LIN {X 0,Y 438.375,Z 352.106,A -85,B 0,C 180,E1 -9180.919,E2 -9180.919} C_VEL
LIN {X 0,Y 438.487,Z 350.298,A -85,B 0,C 180,E1 -9182.756,E2 -9182.756} C_VEL
LIN {X 0,Y 438.587,Z 348.734,A -85,B 0,C 180,E1 -9183.675,E2 -9183.675} C_VEL
LIN {X 0,Y 438.549,Z 345.591,A -85,B 0,C 180,E1 -9185.057,E2 -9185.057} C_VEL
LIN {X 0,Y 438.809,Z 341.362,A -85,B 0,C 180,E1 -9186.437,E2 -9186.437} C_VEL
LIN {X 0,Y 439.034,Z 334.932,A -85,B 0,C 180,E1 -9188.052,E2 -9188.052} C_VEL
LIN {X 0,Y 439.472,Z 327.892,A -85,B 0,C 180,E1 -9189.434,E2 -9189.434} C_VEL
LIN {X 0,Y 439.893,Z 319.12,A -85,B 0,C 180,E1 -9190.82,E2 -9190.82} C_VEL
LIN {X 0,Y 440.436,Z 310.174,A -85,B 0,C 180,E1 -9191.972,E2 -9191.972} C_VEL
LIN {X 0,Y 440.97,Z 299.802,A -85,B 0,C 180,E1 -9193.061,E2 -9193.061} C_VEL
LIN {X 0,Y 441.476,Z 288.11,A -85,B 0,C 180,E1 -9194.05,E2 -9194.05} C_VEL
LIN {X 0,Y 442.042,Z 275.876,A -85,B 0,C 180,E1 -9194.855,E2 -9194.855} C_VEL
LIN {X 0,Y 442.484,Z 263.19,A -85,B 0,C 180,E1 -9195.488,E2 -9195.488} C_VEL
LIN {X 0,Y 440.197,Z 250.38,A -85,B 0,C 180,E1 -9196.025,E2 -9196.025} C_VEL
LIN {X 0,Y 439.232,Z 245.218,A -85,B 0,C 180,E1 -9196.202,E2 -9196.202} C_VEL
LIN {X 0,Y 439.386,Z 236.135,A -85,B 0,C 180,E1 -9199.627,E2 -9199.627} C_VEL
LIN {X 0,Y 439.549,Z 228.372,A -85,B 0,C 180,E1 -9202.566,E2 -9202.566} C_VEL
LIN {X 0,Y 439.72,Z 220.483,A -85,B 0,C 180,E1 -9205.565,E2 -9205.565} C_VEL
LIN {X 0,Y 439.924,Z 212.437,A -85,B 0,C 180,E1 -9208.638,E2 -9208.638} C_VEL
LIN {X 0,Y 440.117,Z 205.533,A -85,B 0,C 180,E1 -9211.264,E2 -9211.264} C_VEL
LIN {X 0,Y 440.24,Z 197.016,A -85,B 0,C 180,E1 -9214.522,E2 -9214.522} C_VEL
LIN {X 0,Y 440.053,Z 192.606,A -85,B 0,C 180,E1 -9216.223,E2 -9216.223} C_VEL
LIN {X 0,Y 439.418,Z 188.752,A -85,B 0,C 180,E1 -9217.79,E2 -9217.79} C_VEL
LIN {X 0,Y 439.381,Z 188.757,A -85,B 0,C 180,E1 -9220.981,E2 -9220.981} C_VEL
LIN {X 0,Y 439.369,Z 188.756,A -85,B 0,C 180,E1 -9223.96,E2 -9223.96} C_VEL
LIN {X 0,Y 439.355,Z 188.756,A -85,B 0,C 180,E1 -9226.54,E2 -9226.54} C_VEL
LIN {X 0,Y 439.386,Z 188.755,A -85,B 0,C 180,E1 -9229.019,E2 -9229.019} C_VEL
